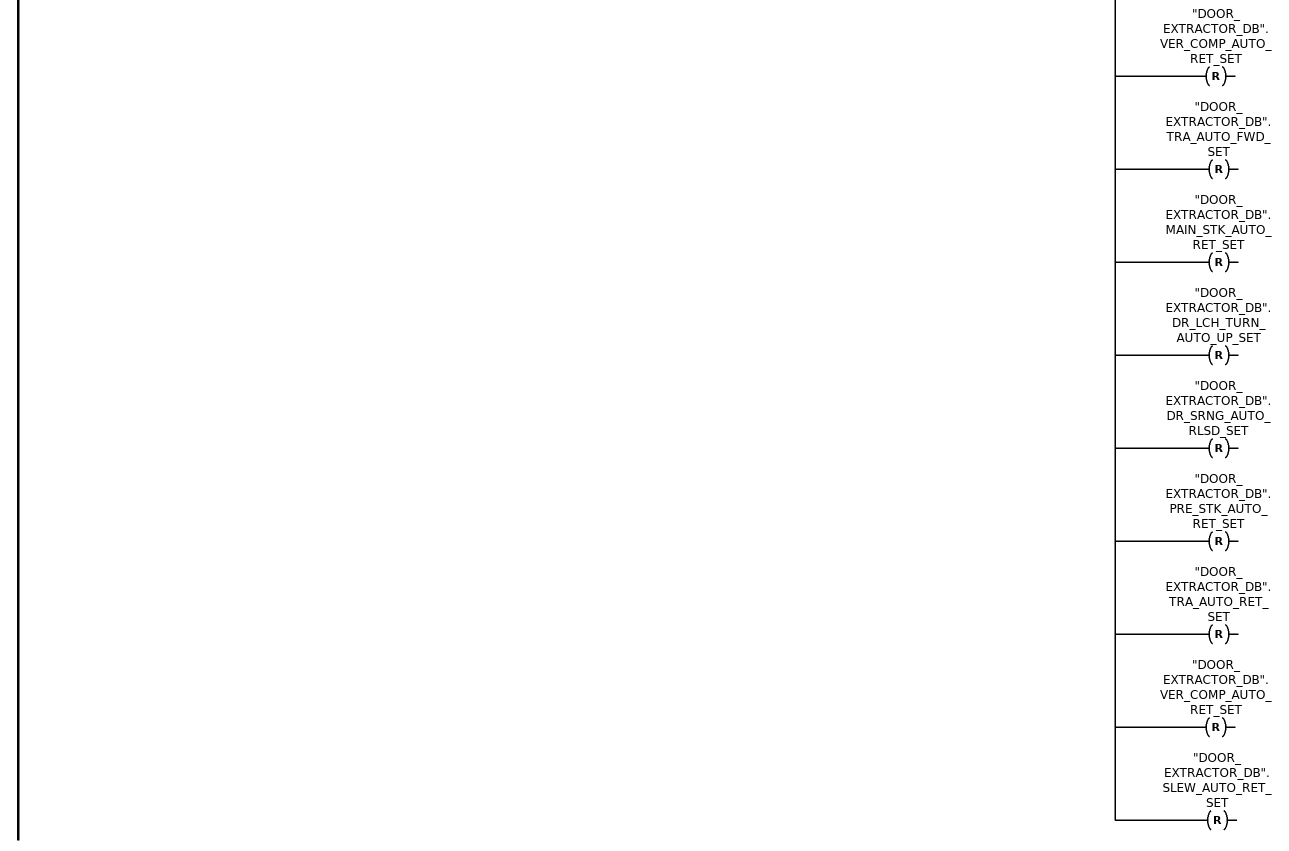
NETWORK
TITLE =
      A     "ALWAYS_ON";
      A     "DOOR_EXTRACTOR_DB".SLEW_NR_FWD_OP_CUT;
      A(;
      O     "DOOR_EXTRACTOR_DB".VER_COMP_RET_OP_CUT;
      O     "ALWAYS_ON";
      );
      A     "DOOR_EXTRACTOR_DB".TRA_NOR_RET_OP_CUT;
      A     "DOOR_EXTRACTOR_DB".PRE_STK_UP_OP_CUT;
      A     "DOOR_EXTRACTOR_DB".DR_SPNG_LK_OP_CUT;
      A     "DOOR_EXTRACTOR_DB".DR_LCH_DN_OP_CUT;
      A     "DOOR_EXTRACTOR_DB".MAIN_STK_UP_OP_CUT;
      A     "DOOR_EXTRACTOR_DB".FIN_STK_UP_OP_CUT;
      =     "DOOR_EXTRACTOR_DB".DR_EXT_AUTO_OPER_FIN;
      R     "DOOR_EXTRACTOR_DB".SLEW_AUTO_FWD_SET;
      R     "DOOR_EXTRACTOR_DB".VER_COMP_AUTO_FWD_SET;
      R     "DOOR_EXTRACTOR_DB".TRA_AUTO_FWD_SET;
      R     "DOOR_EXTRACTOR_DB".PRE_STK_AUTO_FWD_SET;
      R     "DOOR_EXTRACTOR_DB".DR_SPNG_AUTO_PRSD_SET;
      R     "DOOR_EXTRACTOR_DB".DR_LCH_TURN_AUTO_DN_SET;
      R     "DOOR_EXTRACTOR_DB".MAIN_STK_AUTO_FWD_SET;
      R     "DOOR_EXTRACTOR_DB".TRA_AUTO_RET_SET;
      R     "DOOR_EXTRACTOR_DB".VER_COMP_AUTO_RET_SET;
      R     "DOOR_EXTRACTOR_DB".FIN_STK_AUTO_FWD_SET;
      R     "DOOR_EXTRACTOR_DB".SLEW_AUTO_RET_SET;
      R     "DOOR_EXTRACTOR_DB".SLEW_AUTO_FWD_SET;
      R     "DOOR_EXTRACTOR_DB".FIN_STK_AUTO_RET_SET;
      R     "DOOR_EXTRACTOR_DB".VER_COMP_AUTO_RET_SET;
      R     "DOOR_EXTRACTOR_DB".TRA_AUTO_FWD_SET;
      R     "DOOR_EXTRACTOR_DB".MAIN_STK_AUTO_RET_SET;
      R     "DOOR_EXTRACTOR_DB".DR_LCH_TURN_AUTO_UP_SET;
      R     "DOOR_EXTRACTOR_DB".DR_SRNG_AUTO_RLSD_SET;
      R     "DOOR_EXTRACTOR_DB".PRE_STK_AUTO_RET_SET;
      R     "DOOR_EXTRACTOR_DB".TRA_AUTO_RET_SET;
      R     "DOOR_EXTRACTOR_DB".VER_COMP_AUTO_RET_SET;
      R     "DOOR_EXTRACTOR_DB".SLEW_AUTO_RET_SET;
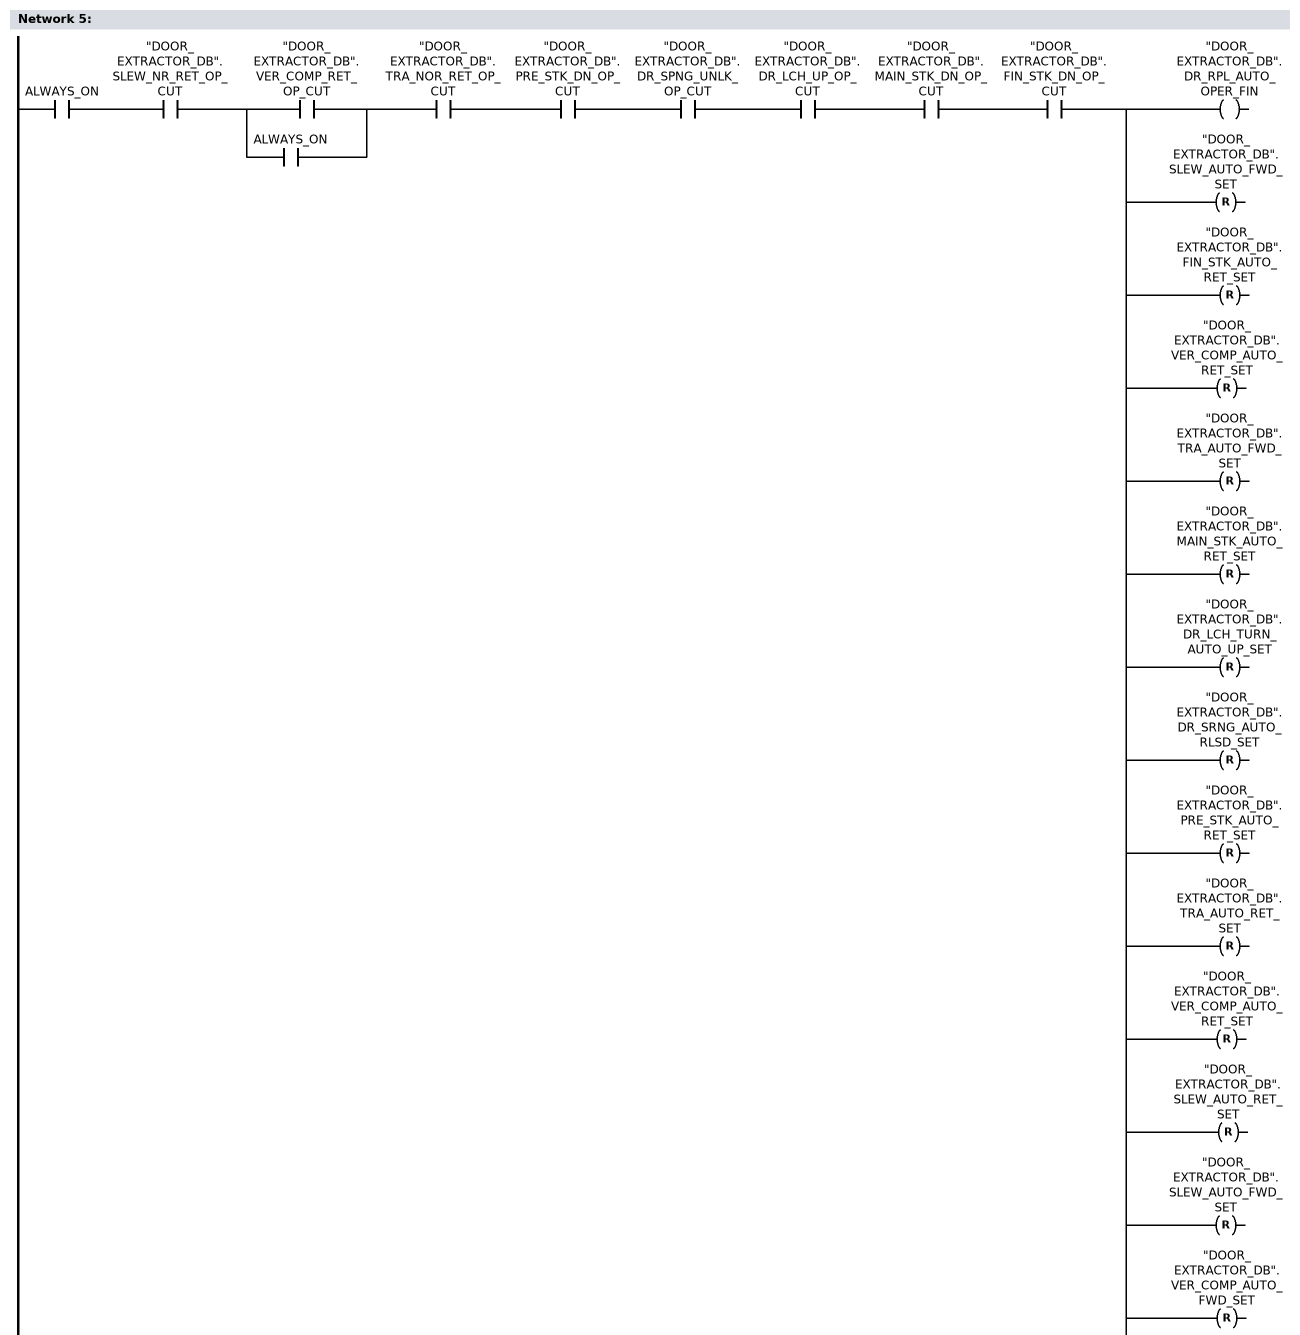
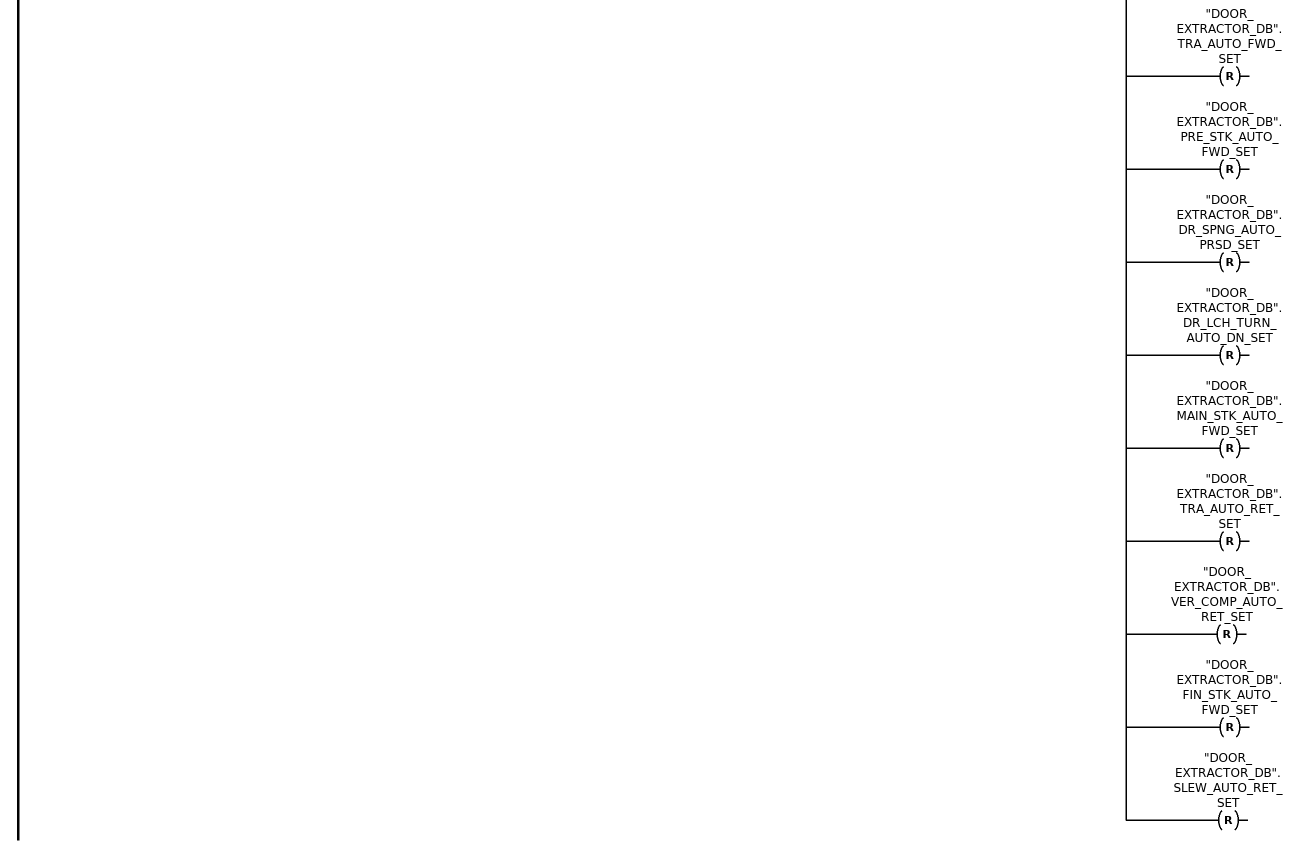
NETWORK
TITLE =
      A     "ALWAYS_ON";
      A     "DOOR_EXTRACTOR_DB".SLEW_NR_RET_OP_CUT;
      A(;
      O     "DOOR_EXTRACTOR_DB".VER_COMP_RET_OP_CUT;
      O     "ALWAYS_ON";
      );
      A     "DOOR_EXTRACTOR_DB".TRA_NOR_RET_OP_CUT;
      A     "DOOR_EXTRACTOR_DB".PRE_STK_DN_OP_CUT;
      A     "DOOR_EXTRACTOR_DB".DR_SPNG_UNLK_OP_CUT;
      A     "DOOR_EXTRACTOR_DB".DR_LCH_UP_OP_CUT;
      A     "DOOR_EXTRACTOR_DB".MAIN_STK_DN_OP_CUT;
      A     "DOOR_EXTRACTOR_DB".FIN_STK_DN_OP_CUT;
      =     "DOOR_EXTRACTOR_DB".DR_RPL_AUTO_OPER_FIN;
      R     "DOOR_EXTRACTOR_DB".SLEW_AUTO_FWD_SET;
      R     "DOOR_EXTRACTOR_DB".FIN_STK_AUTO_RET_SET;
      R     "DOOR_EXTRACTOR_DB".VER_COMP_AUTO_RET_SET;
      R     "DOOR_EXTRACTOR_DB".TRA_AUTO_FWD_SET;
      R     "DOOR_EXTRACTOR_DB".MAIN_STK_AUTO_RET_SET;
      R     "DOOR_EXTRACTOR_DB".DR_LCH_TURN_AUTO_UP_SET;
      R     "DOOR_EXTRACTOR_DB".DR_SRNG_AUTO_RLSD_SET;
      R     "DOOR_EXTRACTOR_DB".PRE_STK_AUTO_RET_SET;
      R     "DOOR_EXTRACTOR_DB".TRA_AUTO_RET_SET;
      R     "DOOR_EXTRACTOR_DB".VER_COMP_AUTO_RET_SET;
      R     "DOOR_EXTRACTOR_DB".SLEW_AUTO_RET_SET;
      R     "DOOR_EXTRACTOR_DB".SLEW_AUTO_FWD_SET;
      R     "DOOR_EXTRACTOR_DB".VER_COMP_AUTO_FWD_SET;
      R     "DOOR_EXTRACTOR_DB".TRA_AUTO_FWD_SET;
      R     "DOOR_EXTRACTOR_DB".PRE_STK_AUTO_FWD_SET;
      R     "DOOR_EXTRACTOR_DB".DR_SPNG_AUTO_PRSD_SET;
      R     "DOOR_EXTRACTOR_DB".DR_LCH_TURN_AUTO_DN_SET;
      R     "DOOR_EXTRACTOR_DB".MAIN_STK_AUTO_FWD_SET;
      R     "DOOR_EXTRACTOR_DB".TRA_AUTO_RET_SET;
      R     "DOOR_EXTRACTOR_DB".VER_COMP_AUTO_RET_SET;
      R     "DOOR_EXTRACTOR_DB".FIN_STK_AUTO_FWD_SET;
      R     "DOOR_EXTRACTOR_DB".SLEW_AUTO_RET_SET;
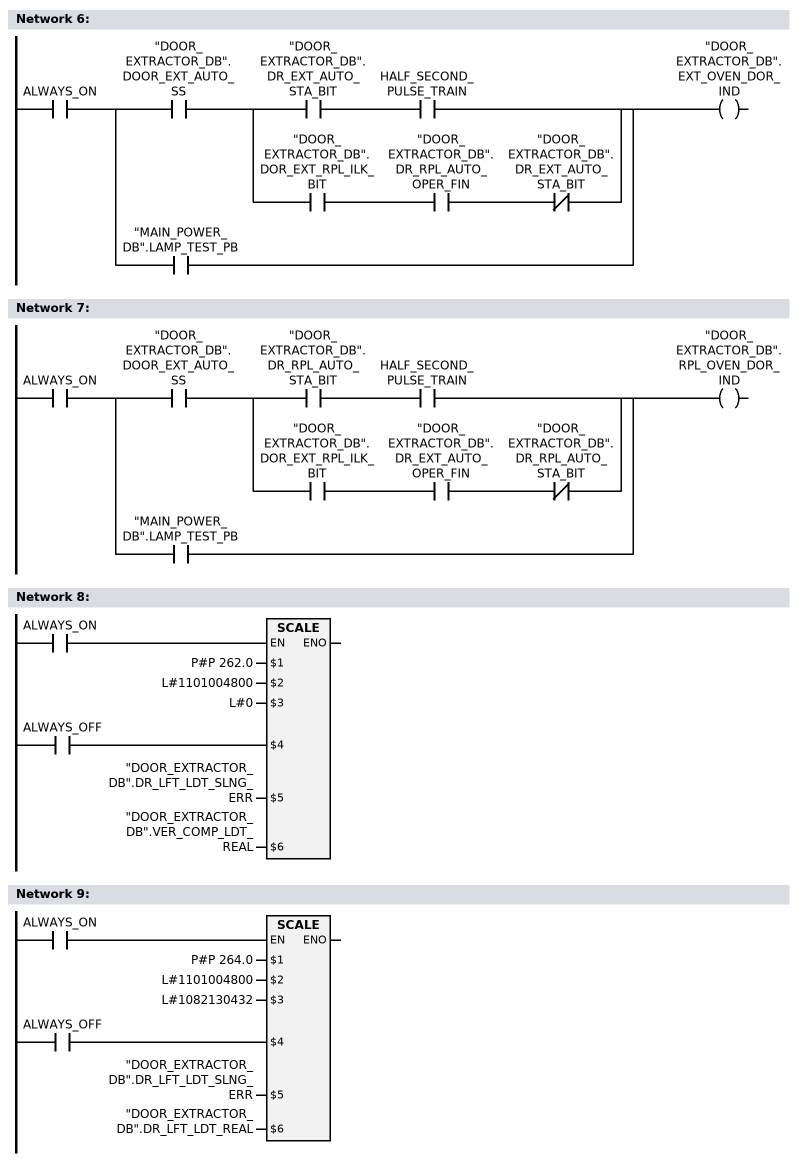
NETWORK
TITLE =
      A     "ALWAYS_ON";
      A(;
      A     "DOOR_EXTRACTOR_DB".DOOR_EXT_AUTO_SS;
      A(;
      A     "DOOR_EXTRACTOR_DB".DR_EXT_AUTO_STA_BIT;
      A     "HALF_SECOND_PULSE_TRAIN";
      O;
      A     "DOOR_EXTRACTOR_DB".DOR_EXT_RPL_ILK_BIT;
      A     "DOOR_EXTRACTOR_DB".DR_RPL_AUTO_OPER_FIN;
      AN    "DOOR_EXTRACTOR_DB".DR_EXT_AUTO_STA_BIT;
      );
      O     "MAIN_POWER_DB".LAMP_TEST_PB;
      );
      =     "DOOR_EXTRACTOR_DB".EXT_OVEN_DOR_IND;
NETWORK
TITLE =
      A     "ALWAYS_ON";
      A(;
      A     "DOOR_EXTRACTOR_DB".DOOR_EXT_AUTO_SS;
      A(;
      A     "DOOR_EXTRACTOR_DB".DR_RPL_AUTO_STA_BIT;
      A     "HALF_SECOND_PULSE_TRAIN";
      O;
      A     "DOOR_EXTRACTOR_DB".DOR_EXT_RPL_ILK_BIT;
      A     "DOOR_EXTRACTOR_DB".DR_EXT_AUTO_OPER_FIN;
      AN    "DOOR_EXTRACTOR_DB".DR_RPL_AUTO_STA_BIT;
      );
      O     "MAIN_POWER_DB".LAMP_TEST_PB;
      );
      =     "DOOR_EXTRACTOR_DB".RPL_OVEN_DOR_IND;
NETWORK
TITLE =
      A     "ALWAYS_OFF";
      =     L 0.0;
      BLD   103;
      A     "ALWAYS_ON";
      JNB   M001;
      CALL  "SCALE" (
           $1                       := P#P 262.0,
           $2                       := L#1101004800,
           $3                       := L#0,
           $4                       := L 0.0,
           $5                       := "DOOR_EXTRACTOR_DB".DR_LFT_LDT_SLNG_ERR,
           $6                       := "DOOR_EXTRACTOR_DB".VER_COMP_LDT_REAL);
M001: NOP   0;
NETWORK
TITLE =
      A     "ALWAYS_OFF";
      =     L 0.0;
      BLD   103;
      A     "ALWAYS_ON";
      JNB   M002;
      CALL  "SCALE" (
           $1                       := P#P 264.0,
           $2                       := L#1101004800,
           $3                       := L#1082130432,
           $4                       := L 0.0,
           $5                       := "DOOR_EXTRACTOR_DB".DR_LFT_LDT_SLNG_ERR,
           $6                       := "DOOR_EXTRACTOR_DB".DR_LFT_LDT_REAL);
M002: NOP   0;
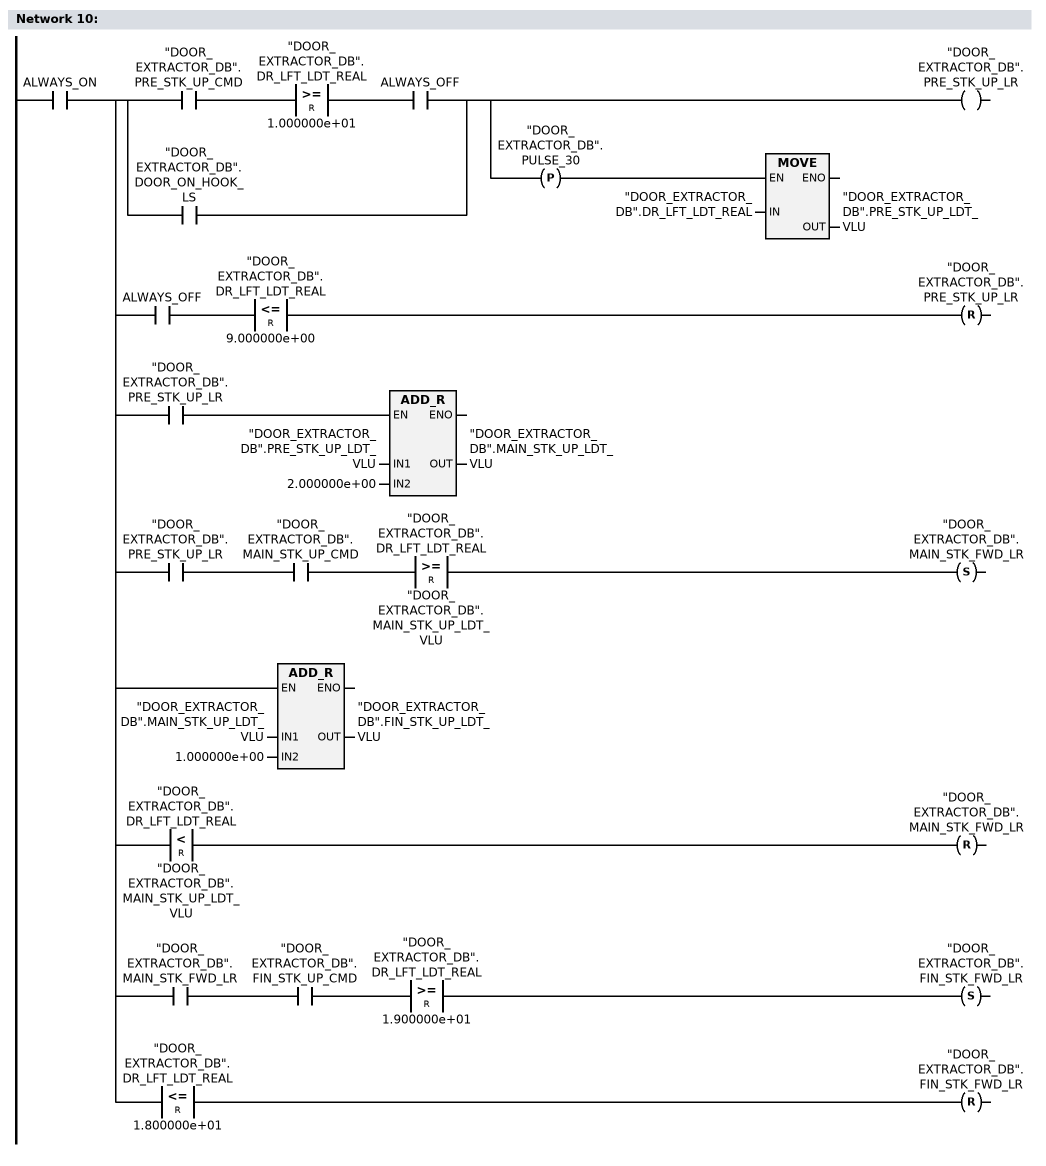
NETWORK
TITLE =
      A     "ALWAYS_ON";
      =     L 0.0;
      A     L 0.0;
      A(;
      A     "DOOR_EXTRACTOR_DB".PRE_STK_UP_CMD;
      A(;
      L     "DOOR_EXTRACTOR_DB".DR_LFT_LDT_REAL;
      L     1.000000e+01;
      >=R;
      );
      A     "ALWAYS_OFF";
      O     "DOOR_EXTRACTOR_DB".DOOR_ON_HOOK_LS;
      );
      =     L 0.1;
      A     L 0.1;
      BLD   102;
      =     "DOOR_EXTRACTOR_DB".PRE_STK_UP_LR;
      A     L 0.1;
      FP    "DOOR_EXTRACTOR_DB".PULSE_30;
      JNB   M003;
      L     "DOOR_EXTRACTOR_DB".DR_LFT_LDT_REAL;
      T     "DOOR_EXTRACTOR_DB".PRE_STK_UP_LDT_VLU;
M003: NOP   0;
      A     L 0.0;
      A     "ALWAYS_OFF";
      A(;
      L     "DOOR_EXTRACTOR_DB".DR_LFT_LDT_REAL;
      L     9.000000e+00;
      <=R;
      );
      R     "DOOR_EXTRACTOR_DB".PRE_STK_UP_LR;
      A     L 0.0;
      A     "DOOR_EXTRACTOR_DB".PRE_STK_UP_LR;
      JNB   M004;
      L     "DOOR_EXTRACTOR_DB".PRE_STK_UP_LDT_VLU;
      L     2.000000e+00;
      +R;
      T     "DOOR_EXTRACTOR_DB".MAIN_STK_UP_LDT_VLU;
M004: NOP   0;
      A     L 0.0;
      A     "DOOR_EXTRACTOR_DB".PRE_STK_UP_LR;
      A     "DOOR_EXTRACTOR_DB".MAIN_STK_UP_CMD;
      A(;
      L     "DOOR_EXTRACTOR_DB".DR_LFT_LDT_REAL;
      L     "DOOR_EXTRACTOR_DB".MAIN_STK_UP_LDT_VLU;
      >=R;
      );
      S     "DOOR_EXTRACTOR_DB".MAIN_STK_FWD_LR;
      A     L 0.0;
      JNB   M005;
      L     "DOOR_EXTRACTOR_DB".MAIN_STK_UP_LDT_VLU;
      L     1.000000e+00;
      +R;
      T     "DOOR_EXTRACTOR_DB".FIN_STK_UP_LDT_VLU;
M005: NOP   0;
      A     L 0.0;
      A(;
      L     "DOOR_EXTRACTOR_DB".DR_LFT_LDT_REAL;
      L     "DOOR_EXTRACTOR_DB".MAIN_STK_UP_LDT_VLU;
      <R;
      );
      R     "DOOR_EXTRACTOR_DB".MAIN_STK_FWD_LR;
      A     L 0.0;
      A     "DOOR_EXTRACTOR_DB".MAIN_STK_FWD_LR;
      A     "DOOR_EXTRACTOR_DB".FIN_STK_UP_CMD;
      A(;
      L     "DOOR_EXTRACTOR_DB".DR_LFT_LDT_REAL;
      L     1.900000e+01;
      >=R;
      );
      S     "DOOR_EXTRACTOR_DB".FIN_STK_FWD_LR;
      A     L 0.0;
      A(;
      L     "DOOR_EXTRACTOR_DB".DR_LFT_LDT_REAL;
      L     1.800000e+01;
      <=R;
      );
      R     "DOOR_EXTRACTOR_DB".FIN_STK_FWD_LR;
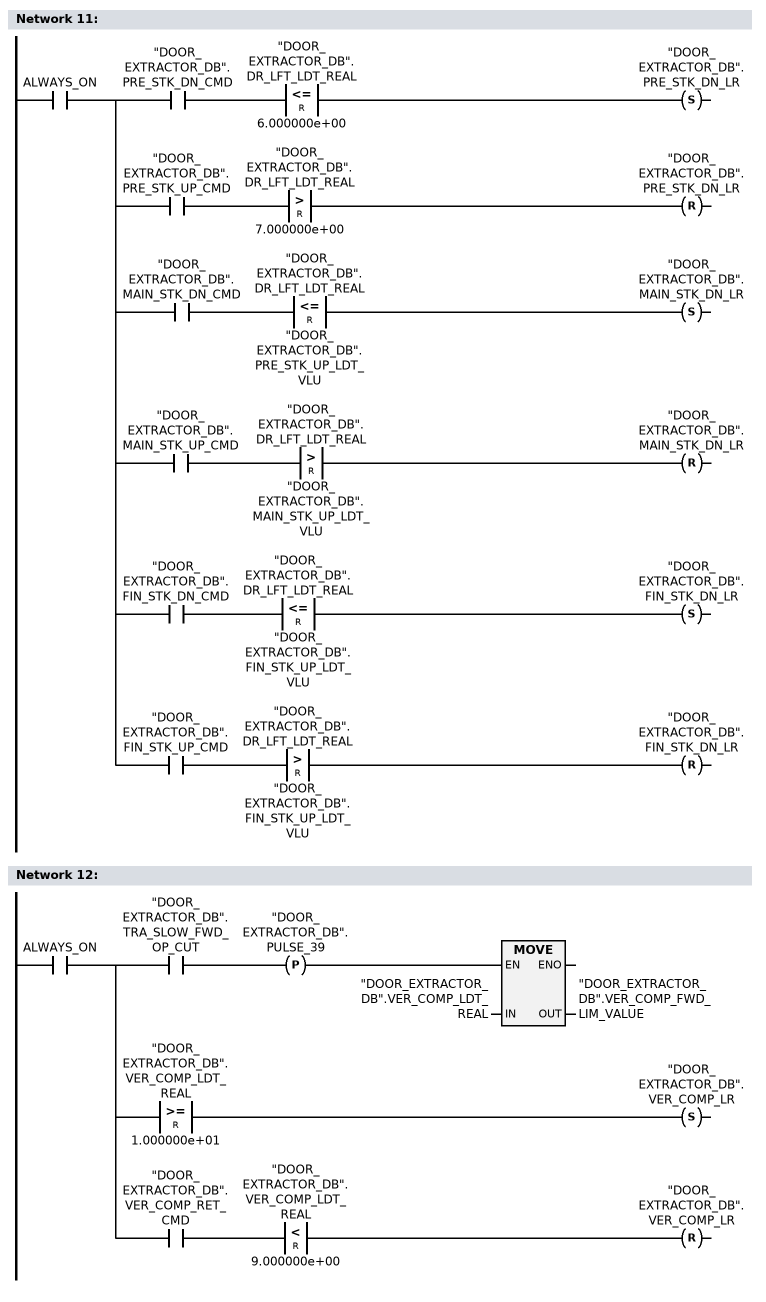
NETWORK
TITLE =
      A     "ALWAYS_ON";
      =     L 0.0;
      A     L 0.0;
      A     "DOOR_EXTRACTOR_DB".PRE_STK_DN_CMD;
      A(;
      L     "DOOR_EXTRACTOR_DB".DR_LFT_LDT_REAL;
      L     6.000000e+00;
      <=R;
      );
      S     "DOOR_EXTRACTOR_DB".PRE_STK_DN_LR;
      A     L 0.0;
      A     "DOOR_EXTRACTOR_DB".PRE_STK_UP_CMD;
      A(;
      L     "DOOR_EXTRACTOR_DB".DR_LFT_LDT_REAL;
      L     7.000000e+00;
      >R;
      );
      R     "DOOR_EXTRACTOR_DB".PRE_STK_DN_LR;
      A     L 0.0;
      A     "DOOR_EXTRACTOR_DB".MAIN_STK_DN_CMD;
      A(;
      L     "DOOR_EXTRACTOR_DB".DR_LFT_LDT_REAL;
      L     "DOOR_EXTRACTOR_DB".PRE_STK_UP_LDT_VLU;
      <=R;
      );
      S     "DOOR_EXTRACTOR_DB".MAIN_STK_DN_LR;
      A     L 0.0;
      A     "DOOR_EXTRACTOR_DB".MAIN_STK_UP_CMD;
      A(;
      L     "DOOR_EXTRACTOR_DB".DR_LFT_LDT_REAL;
      L     "DOOR_EXTRACTOR_DB".MAIN_STK_UP_LDT_VLU;
      >R;
      );
      R     "DOOR_EXTRACTOR_DB".MAIN_STK_DN_LR;
      A     L 0.0;
      A     "DOOR_EXTRACTOR_DB".FIN_STK_DN_CMD;
      A(;
      L     "DOOR_EXTRACTOR_DB".DR_LFT_LDT_REAL;
      L     "DOOR_EXTRACTOR_DB".FIN_STK_UP_LDT_VLU;
      <=R;
      );
      S     "DOOR_EXTRACTOR_DB".FIN_STK_DN_LR;
      A     L 0.0;
      A     "DOOR_EXTRACTOR_DB".FIN_STK_UP_CMD;
      A(;
      L     "DOOR_EXTRACTOR_DB".DR_LFT_LDT_REAL;
      L     "DOOR_EXTRACTOR_DB".FIN_STK_UP_LDT_VLU;
      >R;
      );
      R     "DOOR_EXTRACTOR_DB".FIN_STK_DN_LR;
NETWORK
TITLE =
      A     "ALWAYS_ON";
      =     L 0.0;
      A     L 0.0;
      A     "DOOR_EXTRACTOR_DB".TRA_SLOW_FWD_OP_CUT;
      FP    "DOOR_EXTRACTOR_DB".PULSE_39;
      JNB   M006;
      L     "DOOR_EXTRACTOR_DB".VER_COMP_LDT_REAL;
      T     "DOOR_EXTRACTOR_DB".VER_COMP_FWD_LIM_VALUE;
M006: NOP   0;
      A     L 0.0;
      A(;
      L     "DOOR_EXTRACTOR_DB".VER_COMP_LDT_REAL;
      L     1.000000e+01;
      >=R;
      );
      S     "DOOR_EXTRACTOR_DB".VER_COMP_LR;
      A     L 0.0;
      A     "DOOR_EXTRACTOR_DB".VER_COMP_RET_CMD;
      A(;
      L     "DOOR_EXTRACTOR_DB".VER_COMP_LDT_REAL;
      L     9.000000e+00;
      <R;
      );
      R     "DOOR_EXTRACTOR_DB".VER_COMP_LR;
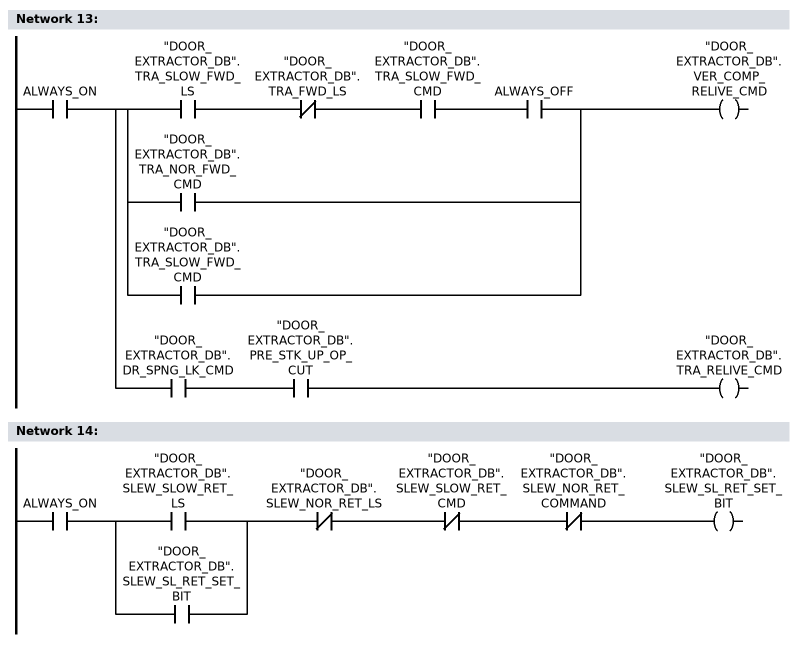
NETWORK
TITLE =
      A     "ALWAYS_ON";
      =     L 0.0;
      A     L 0.0;
      A(;
      A     "DOOR_EXTRACTOR_DB".TRA_SLOW_FWD_LS;
      AN    "DOOR_EXTRACTOR_DB".TRA_FWD_LS;
      A     "DOOR_EXTRACTOR_DB".TRA_SLOW_FWD_CMD;
      A     "ALWAYS_OFF";
      O     "DOOR_EXTRACTOR_DB".TRA_NOR_FWD_CMD;
      O     "DOOR_EXTRACTOR_DB".TRA_SLOW_FWD_CMD;
      );
      =     "DOOR_EXTRACTOR_DB".VER_COMP_RELIVE_CMD;
      A     L 0.0;
      A     "DOOR_EXTRACTOR_DB".DR_SPNG_LK_CMD;
      A     "DOOR_EXTRACTOR_DB".PRE_STK_UP_OP_CUT;
      =     "DOOR_EXTRACTOR_DB".TRA_RELIVE_CMD;
NETWORK
TITLE =
      A     "ALWAYS_ON";
      A(;
      O     "DOOR_EXTRACTOR_DB".SLEW_SLOW_RET_LS;
      O     "DOOR_EXTRACTOR_DB".SLEW_SL_RET_SET_BIT;
      );
      AN    "DOOR_EXTRACTOR_DB".SLEW_NOR_RET_LS;
      AN    "DOOR_EXTRACTOR_DB".SLEW_SLOW_RET_CMD;
      AN    "DOOR_EXTRACTOR_DB".SLEW_NOR_RET_COMMAND;
      =     "DOOR_EXTRACTOR_DB".SLEW_SL_RET_SET_BIT;
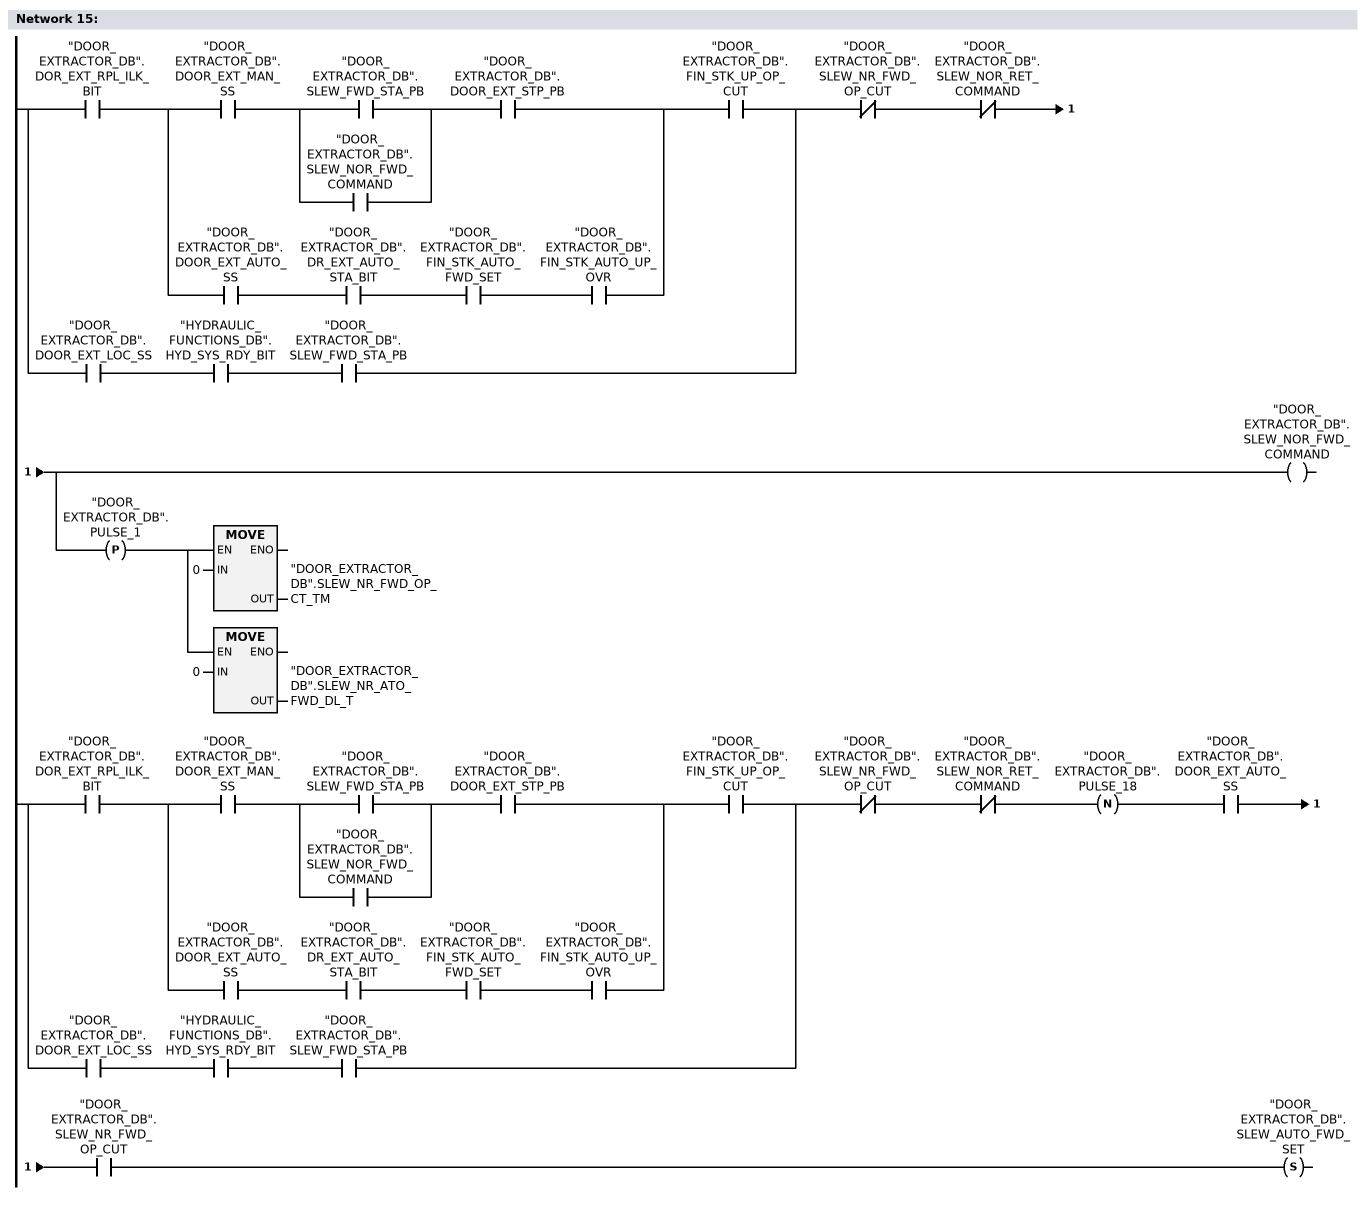
NETWORK
TITLE =
      A(;
      A     "DOOR_EXTRACTOR_DB".DOR_EXT_RPL_ILK_BIT;
      A(;
      A     "DOOR_EXTRACTOR_DB".DOOR_EXT_MAN_SS;
      A(;
      O     "DOOR_EXTRACTOR_DB".SLEW_FWD_STA_PB;
      O     "DOOR_EXTRACTOR_DB".SLEW_NOR_FWD_COMMAND;
      );
      A     "DOOR_EXTRACTOR_DB".DOOR_EXT_STP_PB;
      O;
      A     "DOOR_EXTRACTOR_DB".DOOR_EXT_AUTO_SS;
      A     "DOOR_EXTRACTOR_DB".DR_EXT_AUTO_STA_BIT;
      A     "DOOR_EXTRACTOR_DB".FIN_STK_AUTO_FWD_SET;
      A     "DOOR_EXTRACTOR_DB".FIN_STK_AUTO_UP_OVR;
      );
      A     "DOOR_EXTRACTOR_DB".FIN_STK_UP_OP_CUT;
      O;
      A     "DOOR_EXTRACTOR_DB".DOOR_EXT_LOC_SS;
      A     "HYDRAULIC_FUNCTIONS_DB".HYD_SYS_RDY_BIT;
      A     "DOOR_EXTRACTOR_DB".SLEW_FWD_STA_PB;
      );
      AN    "DOOR_EXTRACTOR_DB".SLEW_NR_FWD_OP_CUT;
      AN    "DOOR_EXTRACTOR_DB".SLEW_NOR_RET_COMMAND;
      =     L 0.0;
      A     L 0.0;
      BLD   102;
      =     "DOOR_EXTRACTOR_DB".SLEW_NOR_FWD_COMMAND;
      A(;
      A     L 0.0;
      FN    "DOOR_EXTRACTOR_DB".PULSE_18;
      );
      A     "DOOR_EXTRACTOR_DB".DOOR_EXT_AUTO_SS;
      A     "DOOR_EXTRACTOR_DB".SLEW_NR_FWD_OP_CUT;
      S     "DOOR_EXTRACTOR_DB".SLEW_AUTO_FWD_SET;
      A     L 0.0;
      FP    "DOOR_EXTRACTOR_DB".PULSE_1;
      =     L 0.1;
      A     L 0.1;
      JNB   M007;
      L     0;
      T     "DOOR_EXTRACTOR_DB".SLEW_NR_FWD_OP_CT_TM;
M007: NOP   0;
      A     L 0.1;
      JNB   M008;
      L     0;
      T     "DOOR_EXTRACTOR_DB".SLEW_NR_ATO_FWD_DL_T;
M008: NOP   0;
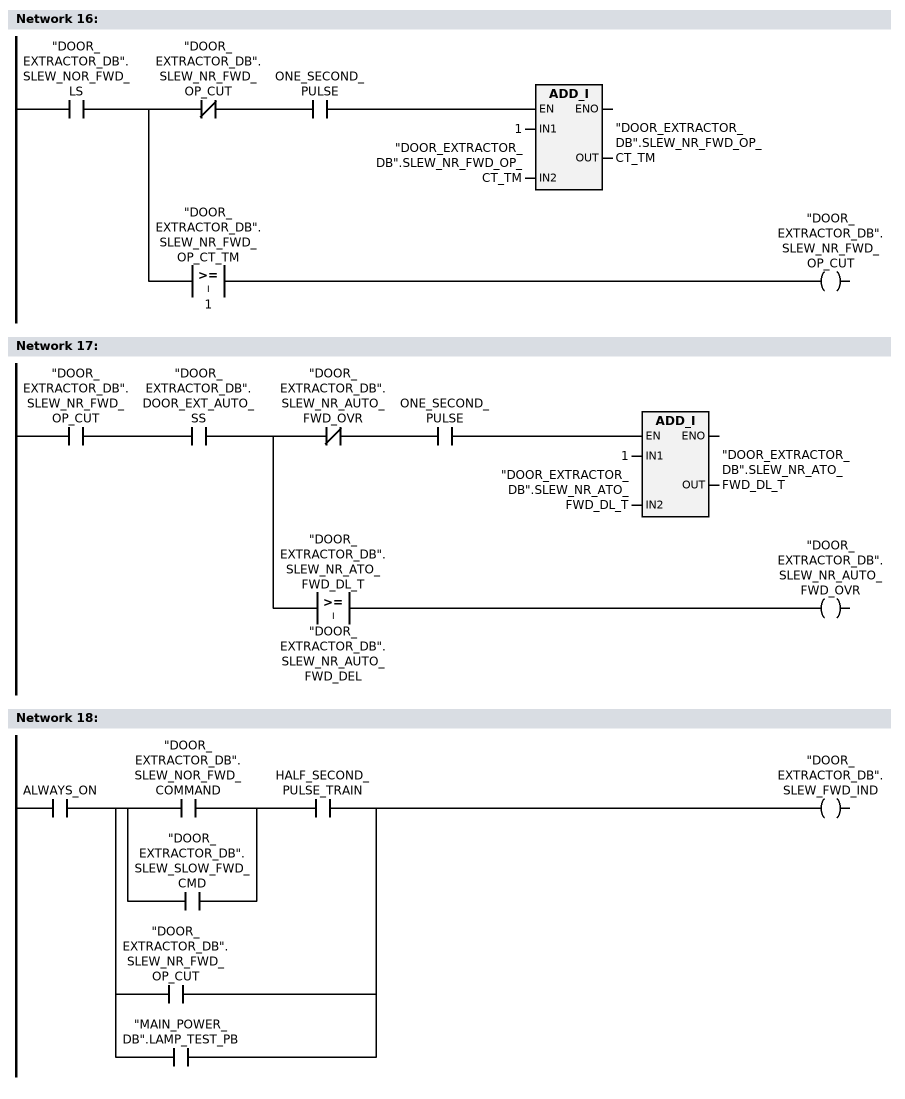
NETWORK
TITLE =
      A     "DOOR_EXTRACTOR_DB".SLEW_NOR_FWD_LS;
      =     L 0.0;
      A     L 0.0;
      AN    "DOOR_EXTRACTOR_DB".SLEW_NR_FWD_OP_CUT;
      A     "ONE_SECOND_PULSE";
      JNB   M009;
      L     1;
      L     "DOOR_EXTRACTOR_DB".SLEW_NR_FWD_OP_CT_TM;
      +I;
      T     "DOOR_EXTRACTOR_DB".SLEW_NR_FWD_OP_CT_TM;
M009: NOP   0;
      A     L 0.0;
      A(;
      L     "DOOR_EXTRACTOR_DB".SLEW_NR_FWD_OP_CT_TM;
      L     1;
      >=I;
      );
      =     "DOOR_EXTRACTOR_DB".SLEW_NR_FWD_OP_CUT;
NETWORK
TITLE =
      A     "DOOR_EXTRACTOR_DB".SLEW_NR_FWD_OP_CUT;
      A     "DOOR_EXTRACTOR_DB".DOOR_EXT_AUTO_SS;
      =     L 0.0;
      A     L 0.0;
      AN    "DOOR_EXTRACTOR_DB".SLEW_NR_AUTO_FWD_OVR;
      A     "ONE_SECOND_PULSE";
      JNB   M010;
      L     1;
      L     "DOOR_EXTRACTOR_DB".SLEW_NR_ATO_FWD_DL_T;
      +I;
      T     "DOOR_EXTRACTOR_DB".SLEW_NR_ATO_FWD_DL_T;
M010: NOP   0;
      A     L 0.0;
      A(;
      L     "DOOR_EXTRACTOR_DB".SLEW_NR_ATO_FWD_DL_T;
      L     "DOOR_EXTRACTOR_DB".SLEW_NR_AUTO_FWD_DEL;
      >=I;
      );
      =     "DOOR_EXTRACTOR_DB".SLEW_NR_AUTO_FWD_OVR;
NETWORK
TITLE =
      A     "ALWAYS_ON";
      A(;
      A(;
      O     "DOOR_EXTRACTOR_DB".SLEW_NOR_FWD_COMMAND;
      O     "DOOR_EXTRACTOR_DB".SLEW_SLOW_FWD_CMD;
      );
      A     "HALF_SECOND_PULSE_TRAIN";
      O     "DOOR_EXTRACTOR_DB".SLEW_NR_FWD_OP_CUT;
      O     "MAIN_POWER_DB".LAMP_TEST_PB;
      );
      =     "DOOR_EXTRACTOR_DB".SLEW_FWD_IND;
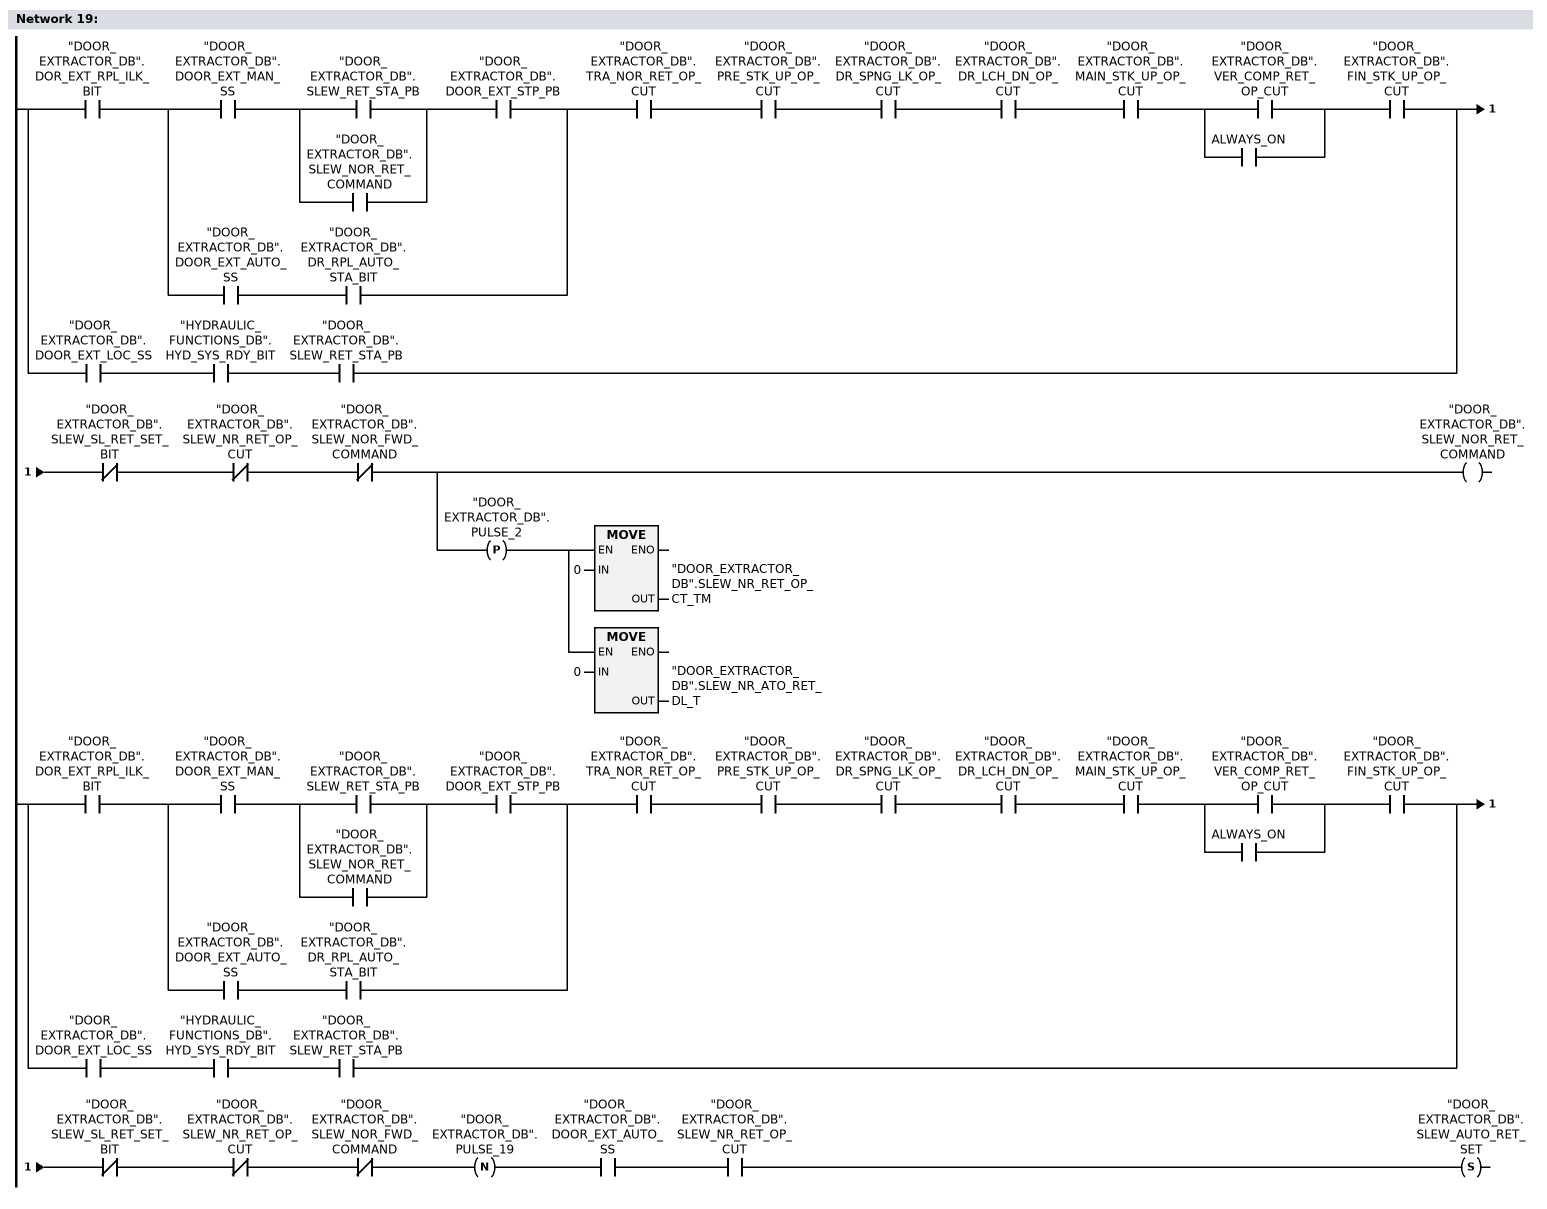
NETWORK
TITLE =
      A(;
      A     "DOOR_EXTRACTOR_DB".DOR_EXT_RPL_ILK_BIT;
      A(;
      A     "DOOR_EXTRACTOR_DB".DOOR_EXT_MAN_SS;
      A(;
      O     "DOOR_EXTRACTOR_DB".SLEW_RET_STA_PB;
      O     "DOOR_EXTRACTOR_DB".SLEW_NOR_RET_COMMAND;
      );
      A     "DOOR_EXTRACTOR_DB".DOOR_EXT_STP_PB;
      O;
      A     "DOOR_EXTRACTOR_DB".DOOR_EXT_AUTO_SS;
      A     "DOOR_EXTRACTOR_DB".DR_RPL_AUTO_STA_BIT;
      );
      A     "DOOR_EXTRACTOR_DB".TRA_NOR_RET_OP_CUT;
      A     "DOOR_EXTRACTOR_DB".PRE_STK_UP_OP_CUT;
      A     "DOOR_EXTRACTOR_DB".DR_SPNG_LK_OP_CUT;
      A     "DOOR_EXTRACTOR_DB".DR_LCH_DN_OP_CUT;
      A     "DOOR_EXTRACTOR_DB".MAIN_STK_UP_OP_CUT;
      A(;
      O     "DOOR_EXTRACTOR_DB".VER_COMP_RET_OP_CUT;
      O     "ALWAYS_ON";
      );
      A     "DOOR_EXTRACTOR_DB".FIN_STK_UP_OP_CUT;
      O;
      A     "DOOR_EXTRACTOR_DB".DOOR_EXT_LOC_SS;
      A     "HYDRAULIC_FUNCTIONS_DB".HYD_SYS_RDY_BIT;
      A     "DOOR_EXTRACTOR_DB".SLEW_RET_STA_PB;
      );
      AN    "DOOR_EXTRACTOR_DB".SLEW_SL_RET_SET_BIT;
      AN    "DOOR_EXTRACTOR_DB".SLEW_NR_RET_OP_CUT;
      AN    "DOOR_EXTRACTOR_DB".SLEW_NOR_FWD_COMMAND;
      =     L 0.0;
      A     L 0.0;
      BLD   102;
      =     "DOOR_EXTRACTOR_DB".SLEW_NOR_RET_COMMAND;
      A(;
      A     L 0.0;
      FN    "DOOR_EXTRACTOR_DB".PULSE_19;
      );
      A     "DOOR_EXTRACTOR_DB".DOOR_EXT_AUTO_SS;
      A     "DOOR_EXTRACTOR_DB".SLEW_NR_RET_OP_CUT;
      S     "DOOR_EXTRACTOR_DB".SLEW_AUTO_RET_SET;
      A     L 0.0;
      FP    "DOOR_EXTRACTOR_DB".PULSE_2;
      =     L 0.1;
      A     L 0.1;
      JNB   M011;
      L     0;
      T     "DOOR_EXTRACTOR_DB".SLEW_NR_RET_OP_CT_TM;
M011: NOP   0;
      A     L 0.1;
      JNB   M012;
      L     0;
      T     "DOOR_EXTRACTOR_DB".SLEW_NR_ATO_RET_DL_T;
M012: NOP   0;
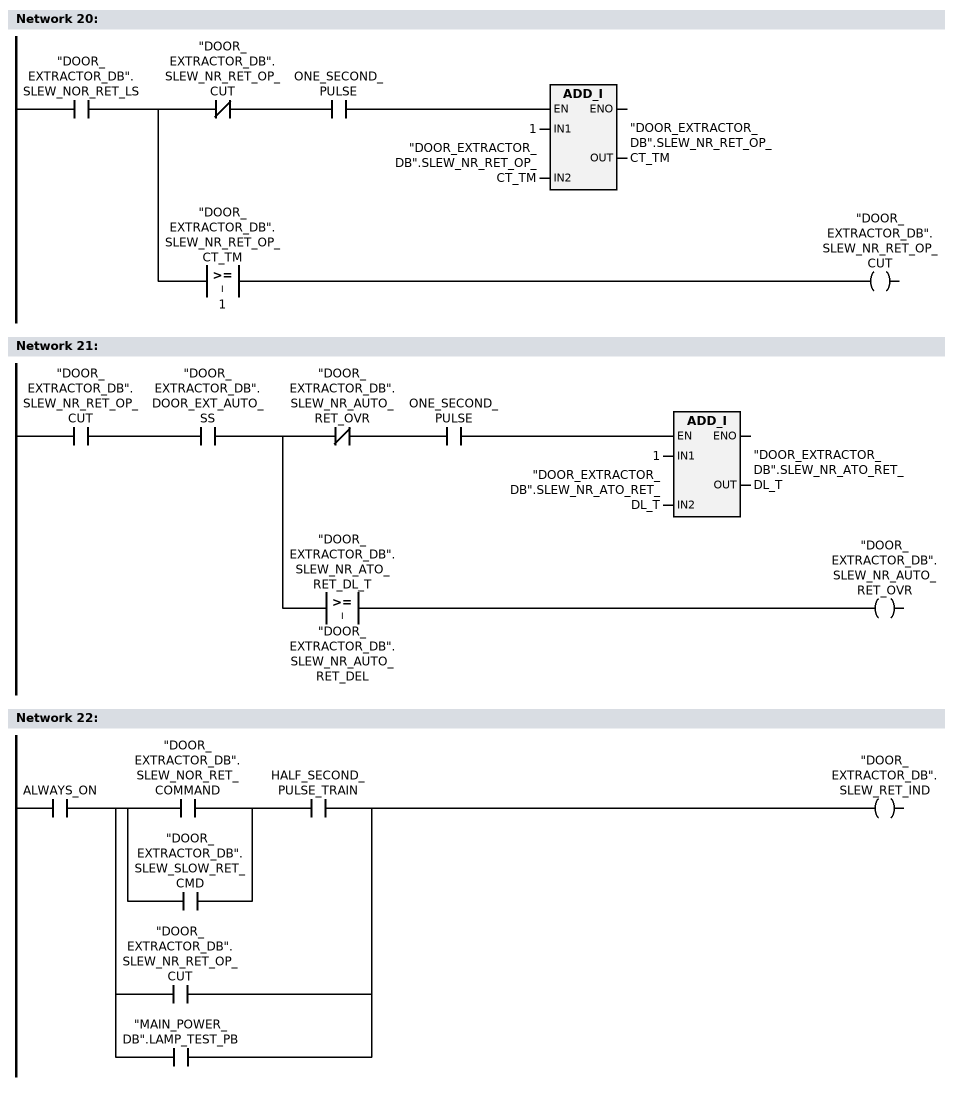
NETWORK
TITLE =
      A     "DOOR_EXTRACTOR_DB".SLEW_NOR_RET_LS;
      =     L 0.0;
      A     L 0.0;
      AN    "DOOR_EXTRACTOR_DB".SLEW_NR_RET_OP_CUT;
      A     "ONE_SECOND_PULSE";
      JNB   M013;
      L     1;
      L     "DOOR_EXTRACTOR_DB".SLEW_NR_RET_OP_CT_TM;
      +I;
      T     "DOOR_EXTRACTOR_DB".SLEW_NR_RET_OP_CT_TM;
M013: NOP   0;
      A     L 0.0;
      A(;
      L     "DOOR_EXTRACTOR_DB".SLEW_NR_RET_OP_CT_TM;
      L     1;
      >=I;
      );
      =     "DOOR_EXTRACTOR_DB".SLEW_NR_RET_OP_CUT;
NETWORK
TITLE =
      A     "DOOR_EXTRACTOR_DB".SLEW_NR_RET_OP_CUT;
      A     "DOOR_EXTRACTOR_DB".DOOR_EXT_AUTO_SS;
      =     L 0.0;
      A     L 0.0;
      AN    "DOOR_EXTRACTOR_DB".SLEW_NR_AUTO_RET_OVR;
      A     "ONE_SECOND_PULSE";
      JNB   M014;
      L     1;
      L     "DOOR_EXTRACTOR_DB".SLEW_NR_ATO_RET_DL_T;
      +I;
      T     "DOOR_EXTRACTOR_DB".SLEW_NR_ATO_RET_DL_T;
M014: NOP   0;
      A     L 0.0;
      A(;
      L     "DOOR_EXTRACTOR_DB".SLEW_NR_ATO_RET_DL_T;
      L     "DOOR_EXTRACTOR_DB".SLEW_NR_AUTO_RET_DEL;
      >=I;
      );
      =     "DOOR_EXTRACTOR_DB".SLEW_NR_AUTO_RET_OVR;
NETWORK
TITLE =
      A     "ALWAYS_ON";
      A(;
      A(;
      O     "DOOR_EXTRACTOR_DB".SLEW_NOR_RET_COMMAND;
      O     "DOOR_EXTRACTOR_DB".SLEW_SLOW_RET_CMD;
      );
      A     "HALF_SECOND_PULSE_TRAIN";
      O     "DOOR_EXTRACTOR_DB".SLEW_NR_RET_OP_CUT;
      O     "MAIN_POWER_DB".LAMP_TEST_PB;
      );
      =     "DOOR_EXTRACTOR_DB".SLEW_RET_IND;
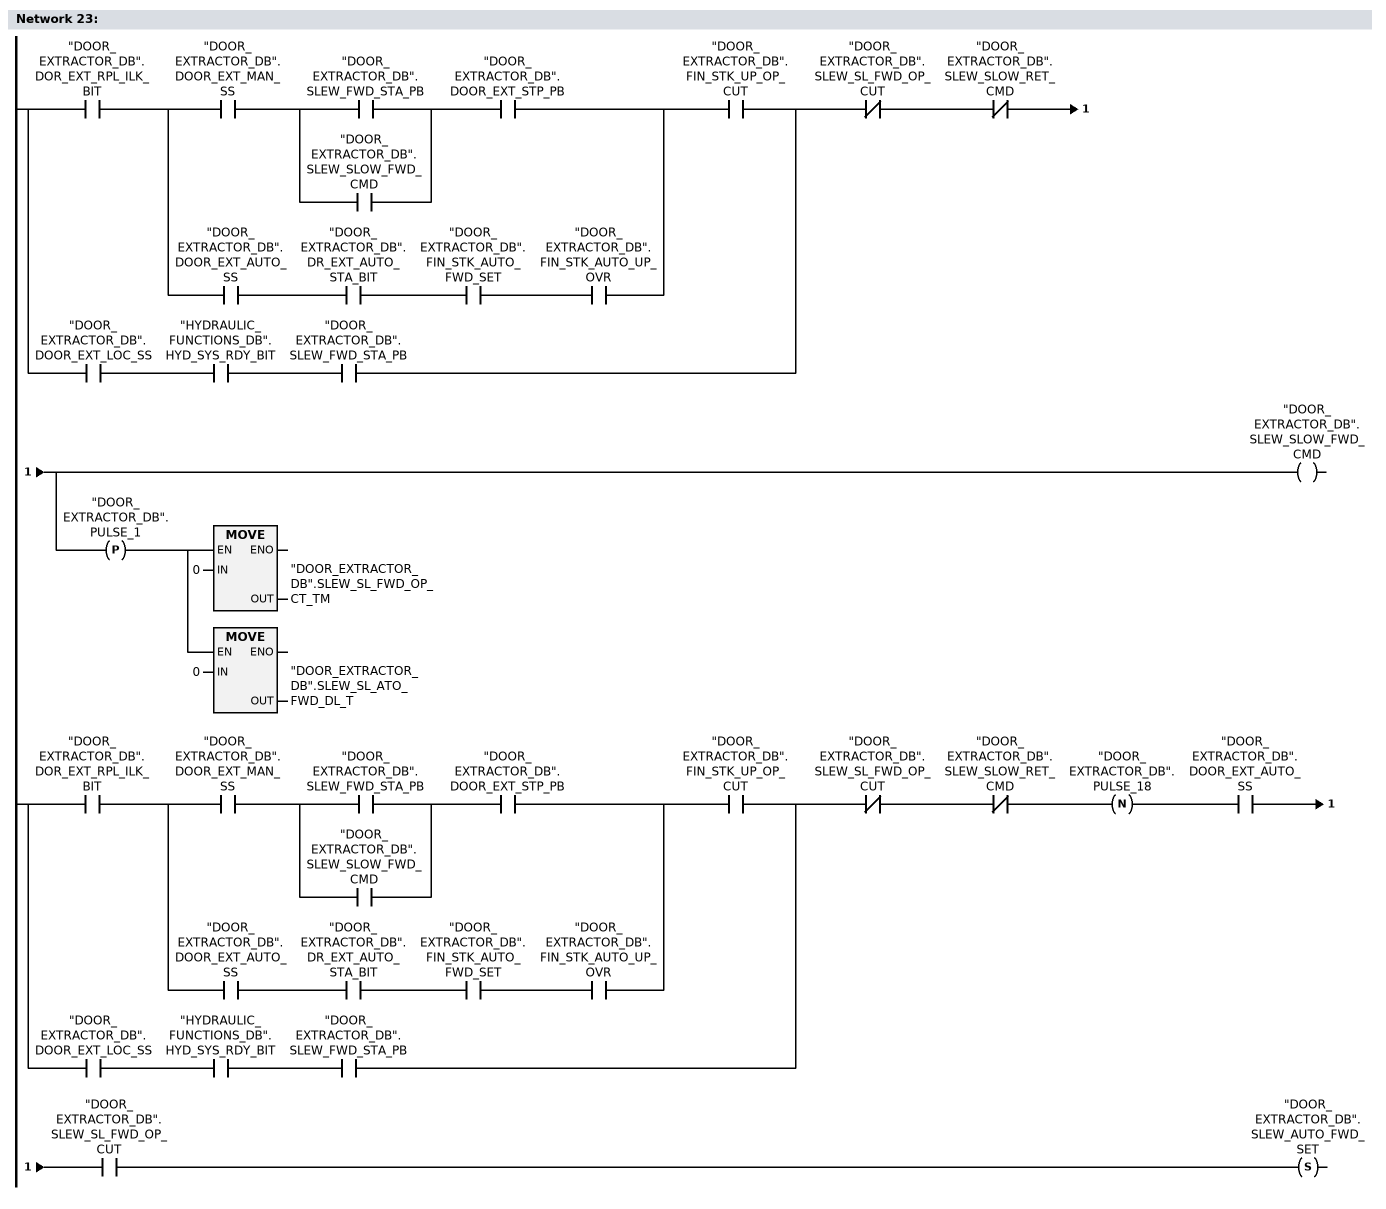
NETWORK
TITLE =
      A(;
      A     "DOOR_EXTRACTOR_DB".DOR_EXT_RPL_ILK_BIT;
      A(;
      A     "DOOR_EXTRACTOR_DB".DOOR_EXT_MAN_SS;
      A(;
      O     "DOOR_EXTRACTOR_DB".SLEW_FWD_STA_PB;
      O     "DOOR_EXTRACTOR_DB".SLEW_SLOW_FWD_CMD;
      );
      A     "DOOR_EXTRACTOR_DB".DOOR_EXT_STP_PB;
      O;
      A     "DOOR_EXTRACTOR_DB".DOOR_EXT_AUTO_SS;
      A     "DOOR_EXTRACTOR_DB".DR_EXT_AUTO_STA_BIT;
      A     "DOOR_EXTRACTOR_DB".FIN_STK_AUTO_FWD_SET;
      A     "DOOR_EXTRACTOR_DB".FIN_STK_AUTO_UP_OVR;
      );
      A     "DOOR_EXTRACTOR_DB".FIN_STK_UP_OP_CUT;
      O;
      A     "DOOR_EXTRACTOR_DB".DOOR_EXT_LOC_SS;
      A     "HYDRAULIC_FUNCTIONS_DB".HYD_SYS_RDY_BIT;
      A     "DOOR_EXTRACTOR_DB".SLEW_FWD_STA_PB;
      );
      AN    "DOOR_EXTRACTOR_DB".SLEW_SL_FWD_OP_CUT;
      AN    "DOOR_EXTRACTOR_DB".SLEW_SLOW_RET_CMD;
      =     L 0.0;
      A     L 0.0;
      BLD   102;
      =     "DOOR_EXTRACTOR_DB".SLEW_SLOW_FWD_CMD;
      A(;
      A     L 0.0;
      FN    "DOOR_EXTRACTOR_DB".PULSE_18;
      );
      A     "DOOR_EXTRACTOR_DB".DOOR_EXT_AUTO_SS;
      A     "DOOR_EXTRACTOR_DB".SLEW_SL_FWD_OP_CUT;
      S     "DOOR_EXTRACTOR_DB".SLEW_AUTO_FWD_SET;
      A     L 0.0;
      FP    "DOOR_EXTRACTOR_DB".PULSE_1;
      =     L 0.1;
      A     L 0.1;
      JNB   M015;
      L     0;
      T     "DOOR_EXTRACTOR_DB".SLEW_SL_FWD_OP_CT_TM;
M015: NOP   0;
      A     L 0.1;
      JNB   M016;
      L     0;
      T     "DOOR_EXTRACTOR_DB".SLEW_SL_ATO_FWD_DL_T;
M016: NOP   0;
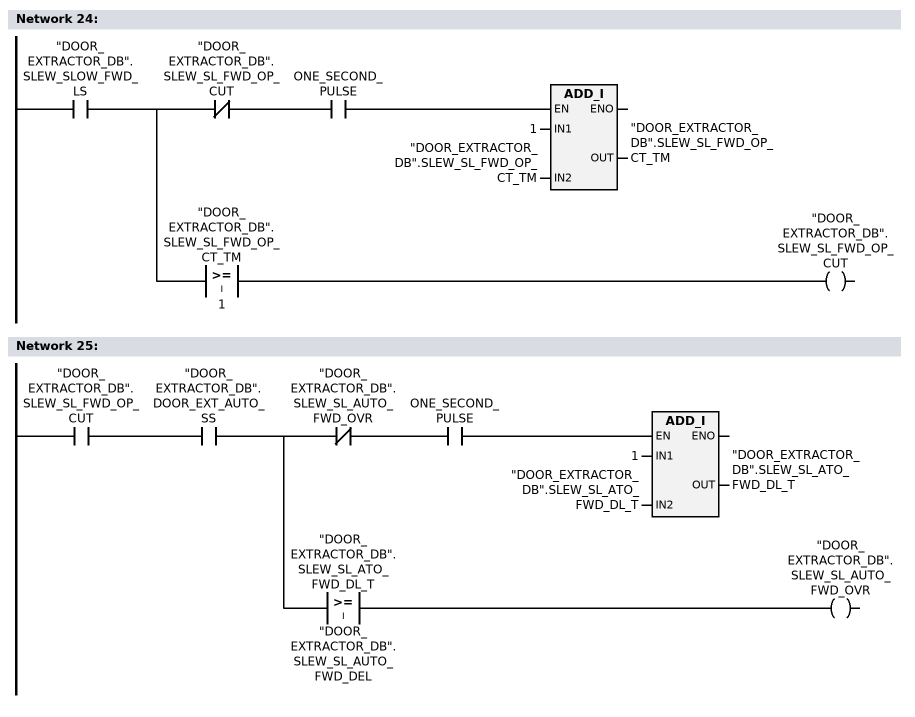
NETWORK
TITLE =
      A     "DOOR_EXTRACTOR_DB".SLEW_SLOW_FWD_LS;
      =     L 0.0;
      A     L 0.0;
      AN    "DOOR_EXTRACTOR_DB".SLEW_SL_FWD_OP_CUT;
      A     "ONE_SECOND_PULSE";
      JNB   M017;
      L     1;
      L     "DOOR_EXTRACTOR_DB".SLEW_SL_FWD_OP_CT_TM;
      +I;
      T     "DOOR_EXTRACTOR_DB".SLEW_SL_FWD_OP_CT_TM;
M017: NOP   0;
      A     L 0.0;
      A(;
      L     "DOOR_EXTRACTOR_DB".SLEW_SL_FWD_OP_CT_TM;
      L     1;
      >=I;
      );
      =     "DOOR_EXTRACTOR_DB".SLEW_SL_FWD_OP_CUT;
NETWORK
TITLE =
      A     "DOOR_EXTRACTOR_DB".SLEW_SL_FWD_OP_CUT;
      A     "DOOR_EXTRACTOR_DB".DOOR_EXT_AUTO_SS;
      =     L 0.0;
      A     L 0.0;
      AN    "DOOR_EXTRACTOR_DB".SLEW_SL_AUTO_FWD_OVR;
      A     "ONE_SECOND_PULSE";
      JNB   M018;
      L     1;
      L     "DOOR_EXTRACTOR_DB".SLEW_SL_ATO_FWD_DL_T;
      +I;
      T     "DOOR_EXTRACTOR_DB".SLEW_SL_ATO_FWD_DL_T;
M018: NOP   0;
      A     L 0.0;
      A(;
      L     "DOOR_EXTRACTOR_DB".SLEW_SL_ATO_FWD_DL_T;
      L     "DOOR_EXTRACTOR_DB".SLEW_SL_AUTO_FWD_DEL;
      >=I;
      );
      =     "DOOR_EXTRACTOR_DB".SLEW_SL_AUTO_FWD_OVR;
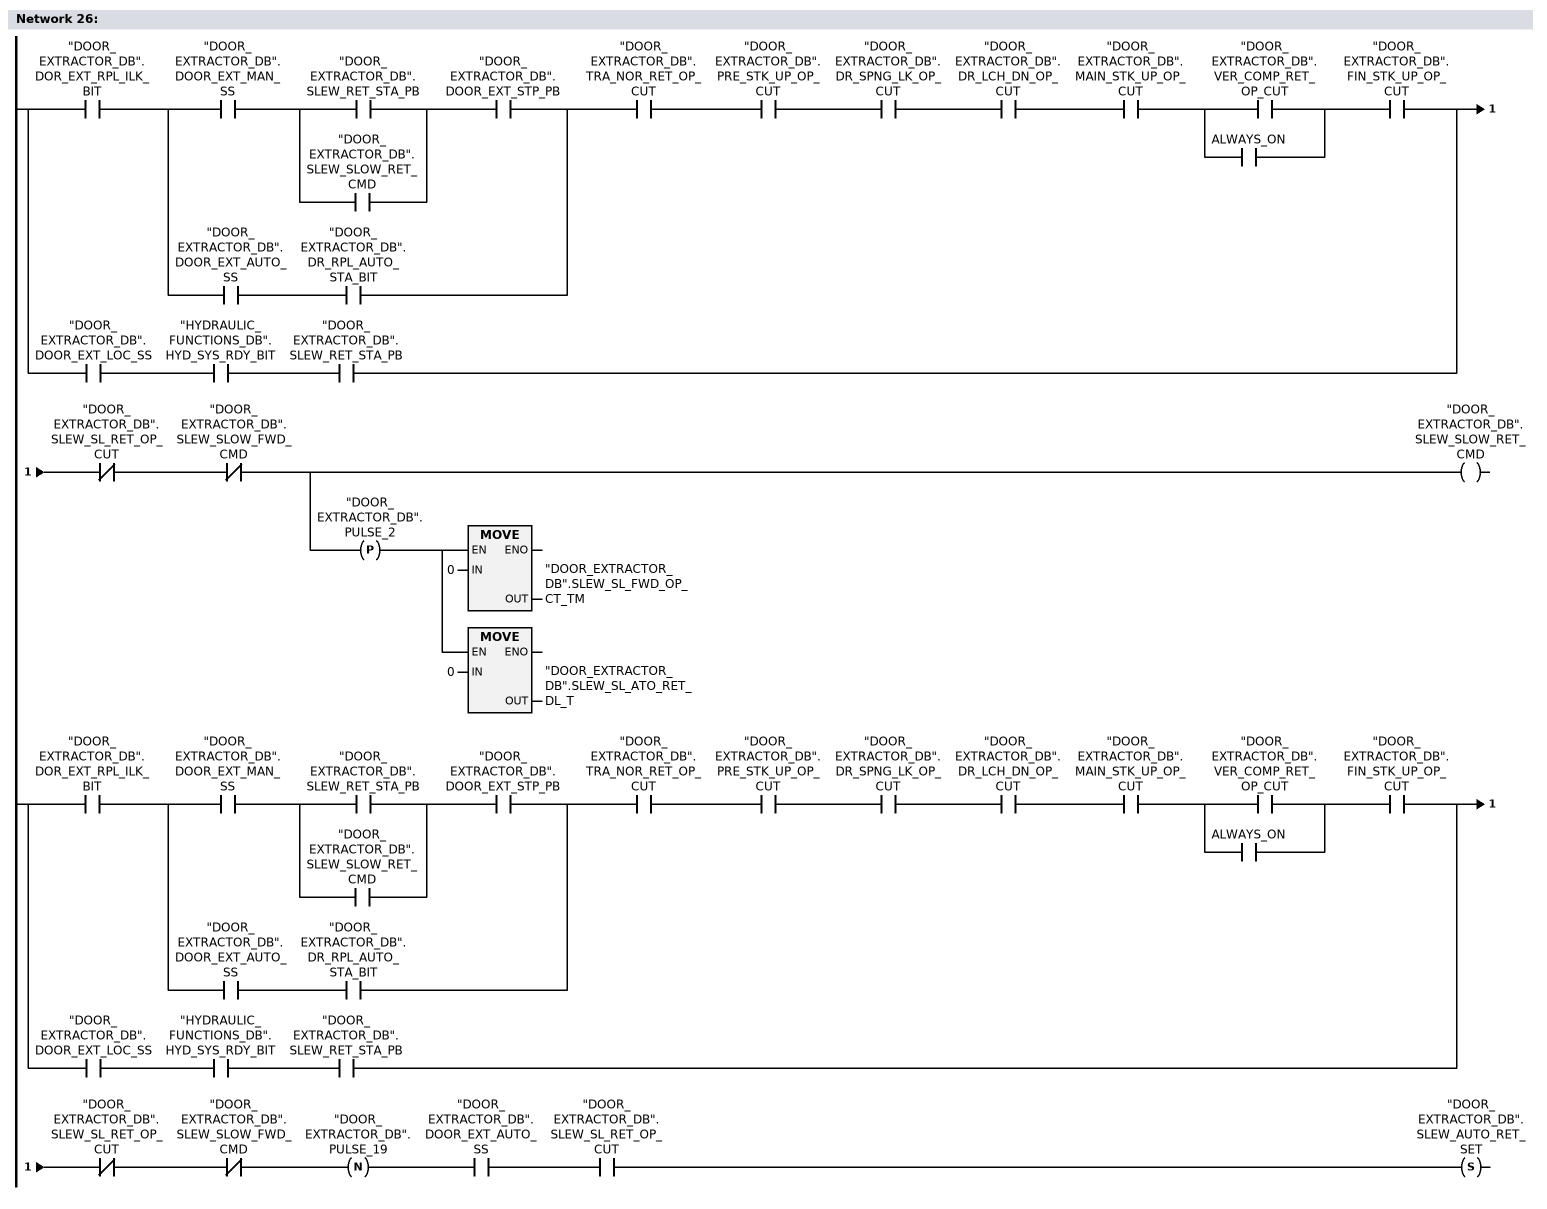
NETWORK
TITLE =
      A(;
      A     "DOOR_EXTRACTOR_DB".DOR_EXT_RPL_ILK_BIT;
      A(;
      A     "DOOR_EXTRACTOR_DB".DOOR_EXT_MAN_SS;
      A(;
      O     "DOOR_EXTRACTOR_DB".SLEW_RET_STA_PB;
      O     "DOOR_EXTRACTOR_DB".SLEW_SLOW_RET_CMD;
      );
      A     "DOOR_EXTRACTOR_DB".DOOR_EXT_STP_PB;
      O;
      A     "DOOR_EXTRACTOR_DB".DOOR_EXT_AUTO_SS;
      A     "DOOR_EXTRACTOR_DB".DR_RPL_AUTO_STA_BIT;
      );
      A     "DOOR_EXTRACTOR_DB".TRA_NOR_RET_OP_CUT;
      A     "DOOR_EXTRACTOR_DB".PRE_STK_UP_OP_CUT;
      A     "DOOR_EXTRACTOR_DB".DR_SPNG_LK_OP_CUT;
      A     "DOOR_EXTRACTOR_DB".DR_LCH_DN_OP_CUT;
      A     "DOOR_EXTRACTOR_DB".MAIN_STK_UP_OP_CUT;
      A(;
      O     "DOOR_EXTRACTOR_DB".VER_COMP_RET_OP_CUT;
      O     "ALWAYS_ON";
      );
      A     "DOOR_EXTRACTOR_DB".FIN_STK_UP_OP_CUT;
      O;
      A     "DOOR_EXTRACTOR_DB".DOOR_EXT_LOC_SS;
      A     "HYDRAULIC_FUNCTIONS_DB".HYD_SYS_RDY_BIT;
      A     "DOOR_EXTRACTOR_DB".SLEW_RET_STA_PB;
      );
      AN    "DOOR_EXTRACTOR_DB".SLEW_SL_RET_OP_CUT;
      AN    "DOOR_EXTRACTOR_DB".SLEW_SLOW_FWD_CMD;
      =     L 0.0;
      A     L 0.0;
      BLD   102;
      =     "DOOR_EXTRACTOR_DB".SLEW_SLOW_RET_CMD;
      A(;
      A     L 0.0;
      FN    "DOOR_EXTRACTOR_DB".PULSE_19;
      );
      A     "DOOR_EXTRACTOR_DB".DOOR_EXT_AUTO_SS;
      A     "DOOR_EXTRACTOR_DB".SLEW_SL_RET_OP_CUT;
      S     "DOOR_EXTRACTOR_DB".SLEW_AUTO_RET_SET;
      A     L 0.0;
      FP    "DOOR_EXTRACTOR_DB".PULSE_2;
      =     L 0.1;
      A     L 0.1;
      JNB   M019;
      L     0;
      T     "DOOR_EXTRACTOR_DB".SLEW_SL_FWD_OP_CT_TM;
M019: NOP   0;
      A     L 0.1;
      JNB   M020;
      L     0;
      T     "DOOR_EXTRACTOR_DB".SLEW_SL_ATO_RET_DL_T;
M020: NOP   0;
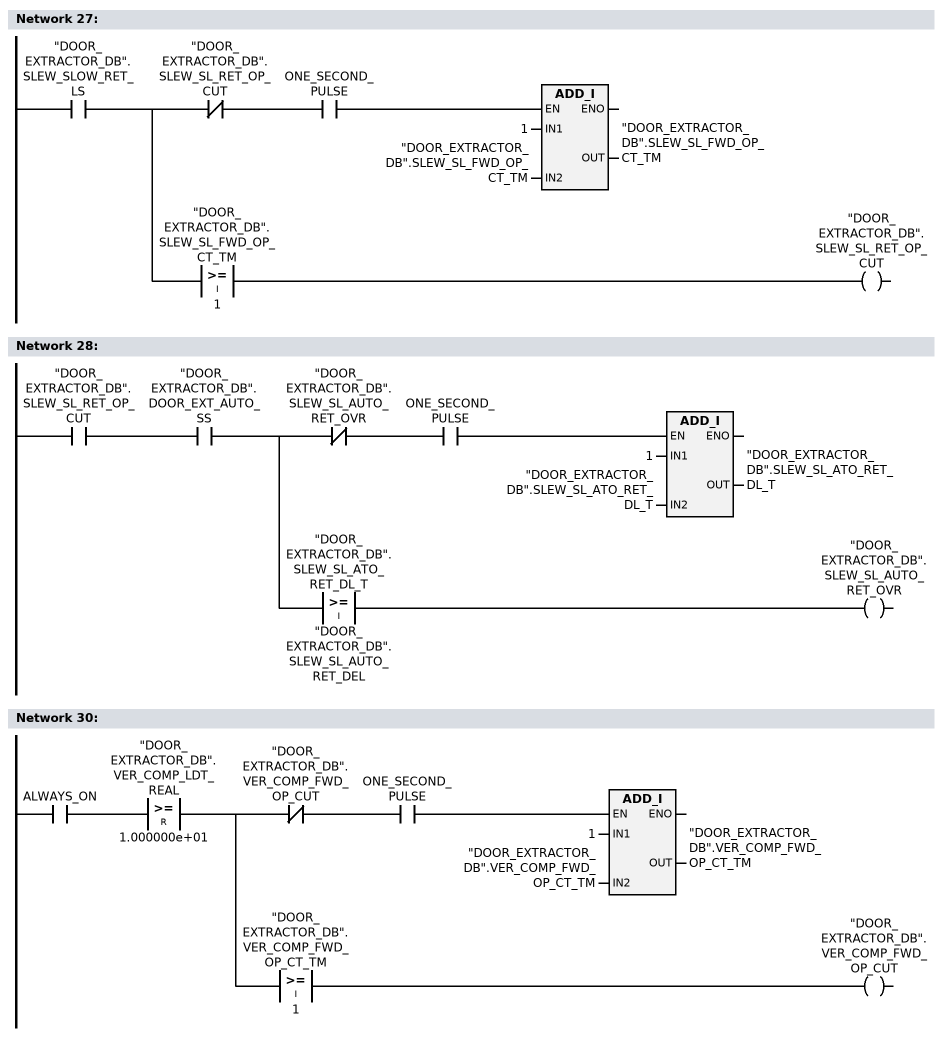
NETWORK
TITLE =
      A     "DOOR_EXTRACTOR_DB".SLEW_SLOW_RET_LS;
      =     L 0.0;
      A     L 0.0;
      AN    "DOOR_EXTRACTOR_DB".SLEW_SL_RET_OP_CUT;
      A     "ONE_SECOND_PULSE";
      JNB   M021;
      L     1;
      L     "DOOR_EXTRACTOR_DB".SLEW_SL_FWD_OP_CT_TM;
      +I;
      T     "DOOR_EXTRACTOR_DB".SLEW_SL_FWD_OP_CT_TM;
M021: NOP   0;
      A     L 0.0;
      A(;
      L     "DOOR_EXTRACTOR_DB".SLEW_SL_FWD_OP_CT_TM;
      L     1;
      >=I;
      );
      =     "DOOR_EXTRACTOR_DB".SLEW_SL_RET_OP_CUT;
NETWORK
TITLE =
      A     "DOOR_EXTRACTOR_DB".SLEW_SL_RET_OP_CUT;
      A     "DOOR_EXTRACTOR_DB".DOOR_EXT_AUTO_SS;
      =     L 0.0;
      A     L 0.0;
      AN    "DOOR_EXTRACTOR_DB".SLEW_SL_AUTO_RET_OVR;
      A     "ONE_SECOND_PULSE";
      JNB   M022;
      L     1;
      L     "DOOR_EXTRACTOR_DB".SLEW_SL_ATO_RET_DL_T;
      +I;
      T     "DOOR_EXTRACTOR_DB".SLEW_SL_ATO_RET_DL_T;
M022: NOP   0;
      A     L 0.0;
      A(;
      L     "DOOR_EXTRACTOR_DB".SLEW_SL_ATO_RET_DL_T;
      L     "DOOR_EXTRACTOR_DB".SLEW_SL_AUTO_RET_DEL;
      >=I;
      );
      =     "DOOR_EXTRACTOR_DB".SLEW_SL_AUTO_RET_OVR;
NETWORK
TITLE =
      A(;
      A     "DOOR_EXTRACTOR_DB".DOR_EXT_RPL_ILK_BIT;
      A(;
      A     "DOOR_EXTRACTOR_DB".DOOR_EXT_MAN_SS;
      A(;
      O     "DOOR_EXTRACTOR_DB".VER_COMP_FWD_STA_PB;
      O     "DOOR_EXTRACTOR_DB".VER_COMP_FWD_CMD;
      );
      A     "DOOR_EXTRACTOR_DB".DOOR_EXT_STP_PB;
      O;
      A     "DOOR_EXTRACTOR_DB".DOOR_EXT_AUTO_SS;
      A(;
      A     "DOOR_EXTRACTOR_DB".DR_EXT_AUTO_STA_BIT;
      A(;
      ON    "DOOR_EXTRACTOR_DB".VER_COMP_AUTO_FWD_SET;
      O     "ALWAYS_ON";
      );
      O;
      A     "DOOR_EXTRACTOR_DB".DR_RPL_AUTO_STA_BIT;
      A     "DOOR_EXTRACTOR_DB".FIN_STK_AUTO_RET_SET;
      A(;
      ON    "DOOR_EXTRACTOR_DB".VER_COMP_AUTO_FWD_SET;
      O     "ALWAYS_ON";
      );
      );
      );
      A(;
      A     "DOOR_EXTRACTOR_DB".SLEW_NR_RET_OP_CUT;
      A     "DOOR_EXTRACTOR_DB".PRE_STK_DN_OP_CUT;
      A     "DOOR_EXTRACTOR_DB".MAIN_STK_DN_OP_CUT;
      A     "DOOR_EXTRACTOR_DB".DR_LCH_UP_OP_CUT;
      A     "DOOR_EXTRACTOR_DB".DR_SPNG_UNLK_OP_CUT;
      O;
      A     "DOOR_EXTRACTOR_DB".SLEW_NR_RET_OP_CUT;
      A     "DOOR_EXTRACTOR_DB".TRA_NOR_RET_OP_CUT;
      A     "DOOR_EXTRACTOR_DB".PRE_STK_UP_OP_CUT;
      A     "DOOR_EXTRACTOR_DB".DR_SPNG_LK_OP_CUT;
      A     "DOOR_EXTRACTOR_DB".DR_LCH_DN_OP_CUT;
      A     "DOOR_EXTRACTOR_DB".MAIN_STK_UP_OP_CUT;
      A     "DOOR_EXTRACTOR_DB".FIN_STK_DN_OP_CUT;
      );
      O;
      A     "DOOR_EXTRACTOR_DB".DOOR_EXT_LOC_SS;
      A     "HYDRAULIC_FUNCTIONS_DB".HYD_SYS_RDY_BIT;
      A     "DOOR_EXTRACTOR_DB".VER_COMP_FWD_STA_PB;
      );
      A(;
      ON    "DOOR_EXTRACTOR_DB".VER_COMP_FWD_OP_CUT;
      O     "ALWAYS_ON";
      );
      AN    "DOOR_EXTRACTOR_DB".VER_COMP_RET_CMD;
      =     L 0.0;
      A     L 0.0;
      AN    "DOOR_EXTRACTOR_DB".DOOR_EXT_AUTO_SS;
      =     L 0.1;
      A     L 0.1;
      BLD   102;
      =     "DOOR_EXTRACTOR_DB".VER_COMP_FWD_CMD;
      A(;
      A     L 0.1;
      FN    "DOOR_EXTRACTOR_DB".PULSE_20;
      );
      A     "DOOR_EXTRACTOR_DB".VER_COMP_FWD_OP_CUT;
      A     "DOOR_EXTRACTOR_DB".DOOR_EXT_AUTO_SS;
      S     "DOOR_EXTRACTOR_DB".VER_COMP_AUTO_FWD_SET;
      A     L 0.0;
      FP    "DOOR_EXTRACTOR_DB".PULSE_3;
      =     L 0.1;
      A     L 0.1;
      A     "DOOR_EXTRACTOR_DB".DOOR_EXT_AUTO_SS;
      S     "DOOR_EXTRACTOR_DB".VER_COMP_AUTO_FWD_SET;
      A     L 0.1;
      JNB   M023;
      L     0;
      T     "DOOR_EXTRACTOR_DB".VER_COMP_FWD_OP_CT_TM;
M023: NOP   0;
      A     L 0.1;
      JNB   M024;
      L     0;
      T     "DOOR_EXTRACTOR_DB".VER_COMP_ATO_FWD_DL_T;
M024: NOP   0;
NETWORK
TITLE =
      A     "ALWAYS_ON";
      A(;
      L     "DOOR_EXTRACTOR_DB".VER_COMP_LDT_REAL;
      L     1.000000e+01;
      >=R;
      );
      =     L 0.0;
      A     L 0.0;
      AN    "DOOR_EXTRACTOR_DB".VER_COMP_FWD_OP_CUT;
      A     "ONE_SECOND_PULSE";
      JNB   M025;
      L     1;
      L     "DOOR_EXTRACTOR_DB".VER_COMP_FWD_OP_CT_TM;
      +I;
      T     "DOOR_EXTRACTOR_DB".VER_COMP_FWD_OP_CT_TM;
M025: NOP   0;
      A     L 0.0;
      A(;
      L     "DOOR_EXTRACTOR_DB".VER_COMP_FWD_OP_CT_TM;
      L     1;
      >=I;
      );
      =     "DOOR_EXTRACTOR_DB".VER_COMP_FWD_OP_CUT;
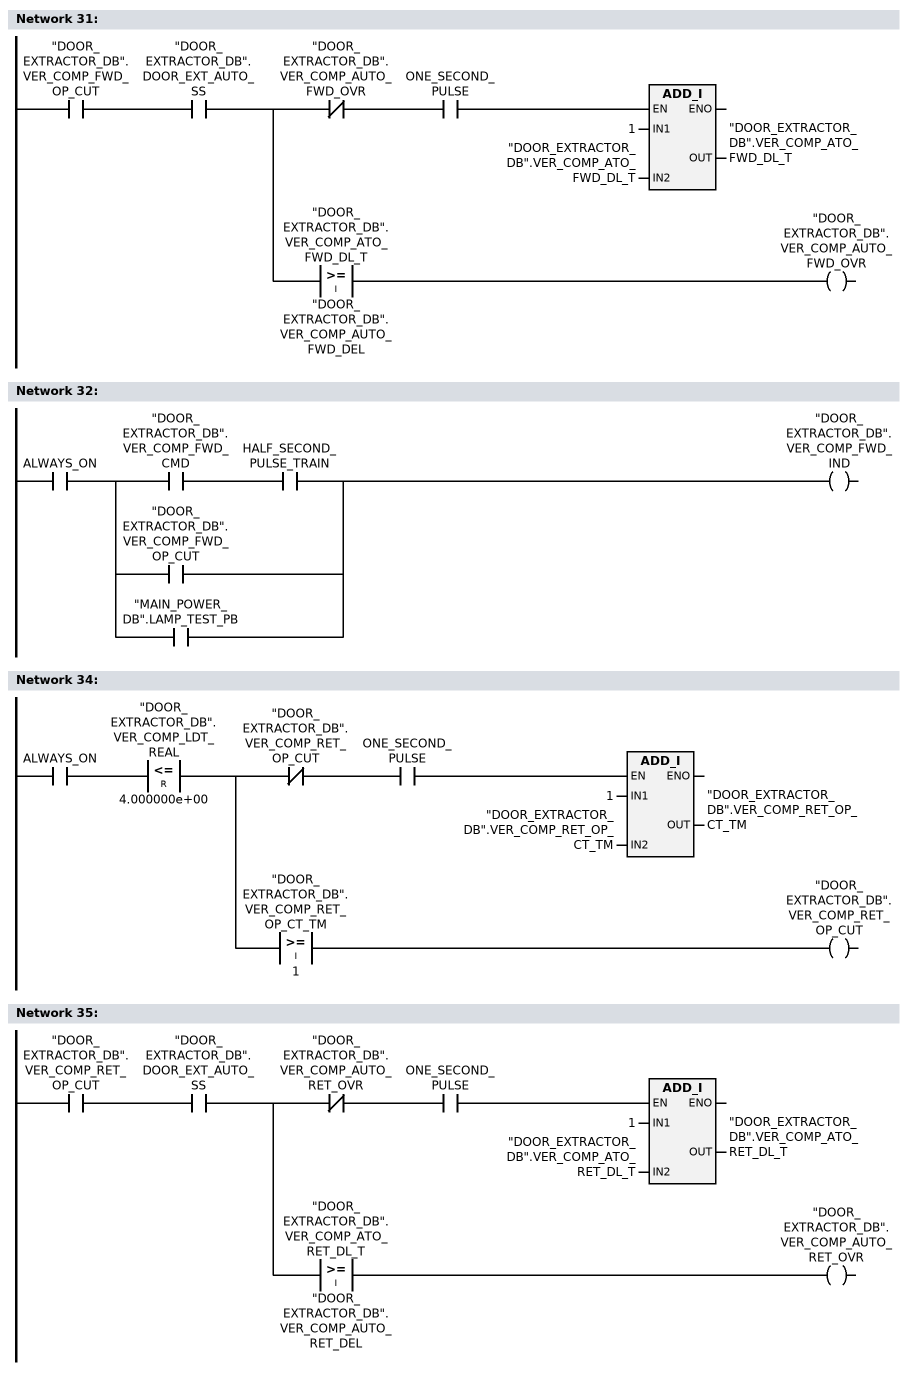
NETWORK
TITLE =
      A     "DOOR_EXTRACTOR_DB".VER_COMP_FWD_OP_CUT;
      A     "DOOR_EXTRACTOR_DB".DOOR_EXT_AUTO_SS;
      =     L 0.0;
      A     L 0.0;
      AN    "DOOR_EXTRACTOR_DB".VER_COMP_AUTO_FWD_OVR;
      A     "ONE_SECOND_PULSE";
      JNB   M026;
      L     1;
      L     "DOOR_EXTRACTOR_DB".VER_COMP_ATO_FWD_DL_T;
      +I;
      T     "DOOR_EXTRACTOR_DB".VER_COMP_ATO_FWD_DL_T;
M026: NOP   0;
      A     L 0.0;
      A(;
      L     "DOOR_EXTRACTOR_DB".VER_COMP_ATO_FWD_DL_T;
      L     "DOOR_EXTRACTOR_DB".VER_COMP_AUTO_FWD_DEL;
      >=I;
      );
      =     "DOOR_EXTRACTOR_DB".VER_COMP_AUTO_FWD_OVR;
NETWORK
TITLE =
      A     "ALWAYS_ON";
      A(;
      A     "DOOR_EXTRACTOR_DB".VER_COMP_FWD_CMD;
      A     "HALF_SECOND_PULSE_TRAIN";
      O     "DOOR_EXTRACTOR_DB".VER_COMP_FWD_OP_CUT;
      O     "MAIN_POWER_DB".LAMP_TEST_PB;
      );
      =     "DOOR_EXTRACTOR_DB".VER_COMP_FWD_IND;
NETWORK
TITLE =
      A(;
      A     "DOOR_EXTRACTOR_DB".DOR_EXT_RPL_ILK_BIT;
      A(;
      A     "DOOR_EXTRACTOR_DB".DOOR_EXT_MAN_SS;
      A(;
      O     "DOOR_EXTRACTOR_DB".VER_COMP_RET_STA_PB;
      O     "DOOR_EXTRACTOR_DB".VER_COMP_RET_CMD;
      );
      A     "DOOR_EXTRACTOR_DB".DOOR_EXT_STP_PB;
      O;
      A     "DOOR_EXTRACTOR_DB".DOOR_EXT_AUTO_SS;
      A(;
      A     "DOOR_EXTRACTOR_DB".DR_EXT_AUTO_STA_BIT;
      A     "DOOR_EXTRACTOR_DB".TRA_AUTO_RET_SET;
      A     "DOOR_EXTRACTOR_DB".TRA_NOR_AUTO_RET_OVR;
      O;
      A     "DOOR_EXTRACTOR_DB".DR_RPL_AUTO_STA_BIT;
      A     "DOOR_EXTRACTOR_DB".TRA_AUTO_RET_SET;
      A     "DOOR_EXTRACTOR_DB".TRA_NOR_AUTO_RET_OVR;
      );
      );
      A(;
      A     "DOOR_EXTRACTOR_DB".SLEW_NR_RET_OP_CUT;
      A     "DOOR_EXTRACTOR_DB".TRA_NOR_RET_OP_CUT;
      A     "DOOR_EXTRACTOR_DB".PRE_STK_UP_OP_CUT;
      A     "DOOR_EXTRACTOR_DB".DR_SPNG_LK_OP_CUT;
      A     "DOOR_EXTRACTOR_DB".DR_LCH_DN_OP_CUT;
      A     "DOOR_EXTRACTOR_DB".MAIN_STK_UP_OP_CUT;
      O;
      A     "DOOR_EXTRACTOR_DB".SLEW_NR_RET_OP_CUT;
      A     "DOOR_EXTRACTOR_DB".TRA_NOR_RET_OP_CUT;
      A     "DOOR_EXTRACTOR_DB".PRE_STK_DN_OP_CUT;
      A     "DOOR_EXTRACTOR_DB".DR_SPNG_UNLK_OP_CUT;
      A     "DOOR_EXTRACTOR_DB".DR_LCH_UP_OP_CUT;
      A     "DOOR_EXTRACTOR_DB".MAIN_STK_DN_OP_CUT;
      A     "DOOR_EXTRACTOR_DB".FIN_STK_DN_OP_CUT;
      );
      O;
      A     "DOOR_EXTRACTOR_DB".DOOR_EXT_LOC_SS;
      A     "HYDRAULIC_FUNCTIONS_DB".HYD_SYS_RDY_BIT;
      A     "DOOR_EXTRACTOR_DB".VER_COMP_RET_STA_PB;
      );
      A(;
      ON    "DOOR_EXTRACTOR_DB".VER_COMP_RET_OP_CUT;
      O     "ALWAYS_ON";
      );
      AN    "DOOR_EXTRACTOR_DB".VER_COMP_FWD_CMD;
      =     L 0.0;
      A     L 0.0;
      AN    "DOOR_EXTRACTOR_DB".DOOR_EXT_AUTO_SS;
      =     L 0.1;
      A     L 0.1;
      BLD   102;
      =     "DOOR_EXTRACTOR_DB".VER_COMP_RET_CMD;
      A(;
      A     L 0.1;
      FN    "DOOR_EXTRACTOR_DB".PULSE_21;
      );
      A     "DOOR_EXTRACTOR_DB".DOOR_EXT_AUTO_SS;
      A     "DOOR_EXTRACTOR_DB".VER_COMP_RET_OP_CUT;
      S     "DOOR_EXTRACTOR_DB".VER_COMP_AUTO_RET_SET;
      A     L 0.0;
      FP    "DOOR_EXTRACTOR_DB".PULSE_4;
      =     L 0.1;
      A     L 0.1;
      A     "DOOR_EXTRACTOR_DB".DOOR_EXT_AUTO_SS;
      S     "DOOR_EXTRACTOR_DB".VER_COMP_AUTO_RET_SET;
      A     L 0.1;
      JNB   M027;
      L     0;
      T     "DOOR_EXTRACTOR_DB".VER_COMP_RET_OP_CT_TM;
M027: NOP   0;
      A     L 0.1;
      JNB   M028;
      L     0;
      T     "DOOR_EXTRACTOR_DB".VER_COMP_ATO_RET_DL_T;
M028: NOP   0;
NETWORK
TITLE =
      A     "ALWAYS_ON";
      A(;
      L     "DOOR_EXTRACTOR_DB".VER_COMP_LDT_REAL;
      L     4.000000e+00;
      <=R;
      );
      =     L 0.0;
      A     L 0.0;
      AN    "DOOR_EXTRACTOR_DB".VER_COMP_RET_OP_CUT;
      A     "ONE_SECOND_PULSE";
      JNB   M029;
      L     1;
      L     "DOOR_EXTRACTOR_DB".VER_COMP_RET_OP_CT_TM;
      +I;
      T     "DOOR_EXTRACTOR_DB".VER_COMP_RET_OP_CT_TM;
M029: NOP   0;
      A     L 0.0;
      A(;
      L     "DOOR_EXTRACTOR_DB".VER_COMP_RET_OP_CT_TM;
      L     1;
      >=I;
      );
      =     "DOOR_EXTRACTOR_DB".VER_COMP_RET_OP_CUT;
NETWORK
TITLE =
      A     "DOOR_EXTRACTOR_DB".VER_COMP_RET_OP_CUT;
      A     "DOOR_EXTRACTOR_DB".DOOR_EXT_AUTO_SS;
      =     L 0.0;
      A     L 0.0;
      AN    "DOOR_EXTRACTOR_DB".VER_COMP_AUTO_RET_OVR;
      A     "ONE_SECOND_PULSE";
      JNB   M030;
      L     1;
      L     "DOOR_EXTRACTOR_DB".VER_COMP_ATO_RET_DL_T;
      +I;
      T     "DOOR_EXTRACTOR_DB".VER_COMP_ATO_RET_DL_T;
M030: NOP   0;
      A     L 0.0;
      A(;
      L     "DOOR_EXTRACTOR_DB".VER_COMP_ATO_RET_DL_T;
      L     "DOOR_EXTRACTOR_DB".VER_COMP_AUTO_RET_DEL;
      >=I;
      );
      =     "DOOR_EXTRACTOR_DB".VER_COMP_AUTO_RET_OVR;
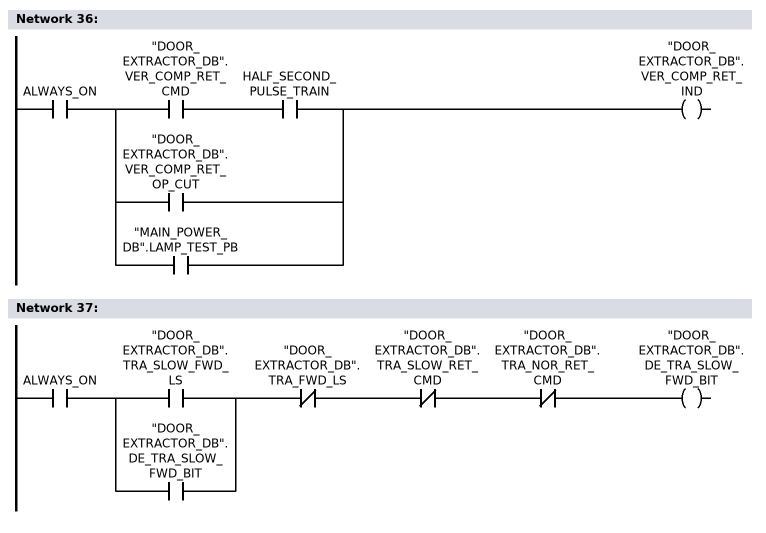
NETWORK
TITLE =
      A     "ALWAYS_ON";
      A(;
      A     "DOOR_EXTRACTOR_DB".VER_COMP_RET_CMD;
      A     "HALF_SECOND_PULSE_TRAIN";
      O     "DOOR_EXTRACTOR_DB".VER_COMP_RET_OP_CUT;
      O     "MAIN_POWER_DB".LAMP_TEST_PB;
      );
      =     "DOOR_EXTRACTOR_DB".VER_COMP_RET_IND;
NETWORK
TITLE =
      A     "ALWAYS_ON";
      A(;
      O     "DOOR_EXTRACTOR_DB".TRA_SLOW_FWD_LS;
      O     "DOOR_EXTRACTOR_DB".DE_TRA_SLOW_FWD_BIT;
      );
      AN    "DOOR_EXTRACTOR_DB".TRA_FWD_LS;
      AN    "DOOR_EXTRACTOR_DB".TRA_SLOW_RET_CMD;
      AN    "DOOR_EXTRACTOR_DB".TRA_NOR_RET_CMD;
      =     "DOOR_EXTRACTOR_DB".DE_TRA_SLOW_FWD_BIT;
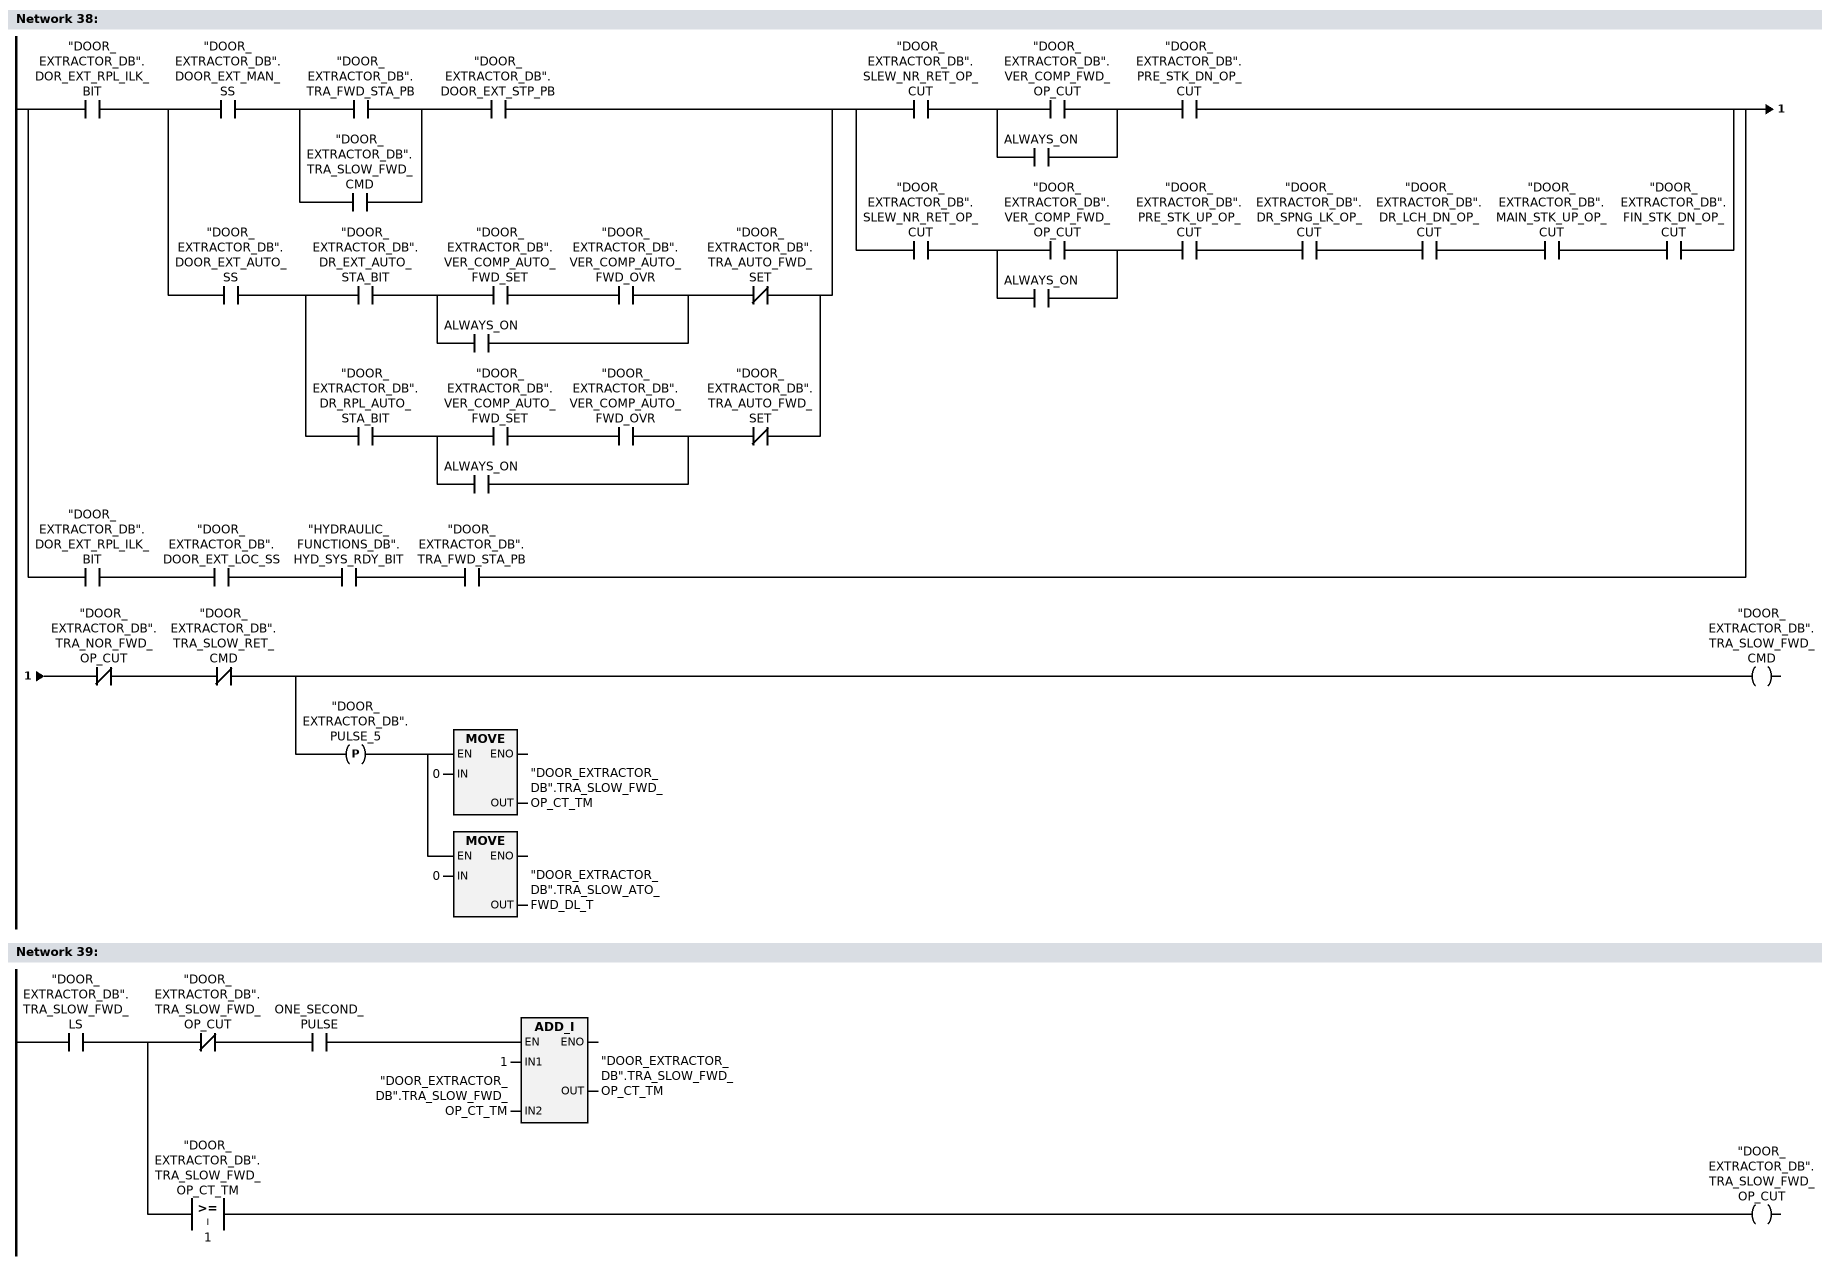
NETWORK
TITLE =
      A(;
      A     "DOOR_EXTRACTOR_DB".DOR_EXT_RPL_ILK_BIT;
      A(;
      A     "DOOR_EXTRACTOR_DB".DOOR_EXT_MAN_SS;
      A(;
      O     "DOOR_EXTRACTOR_DB".TRA_FWD_STA_PB;
      O     "DOOR_EXTRACTOR_DB".TRA_SLOW_FWD_CMD;
      );
      A     "DOOR_EXTRACTOR_DB".DOOR_EXT_STP_PB;
      O;
      A     "DOOR_EXTRACTOR_DB".DOOR_EXT_AUTO_SS;
      A(;
      A     "DOOR_EXTRACTOR_DB".DR_EXT_AUTO_STA_BIT;
      A(;
      A     "DOOR_EXTRACTOR_DB".VER_COMP_AUTO_FWD_SET;
      A     "DOOR_EXTRACTOR_DB".VER_COMP_AUTO_FWD_OVR;
      O     "ALWAYS_ON";
      );
      AN    "DOOR_EXTRACTOR_DB".TRA_AUTO_FWD_SET;
      O;
      A     "DOOR_EXTRACTOR_DB".DR_RPL_AUTO_STA_BIT;
      A(;
      A     "DOOR_EXTRACTOR_DB".VER_COMP_AUTO_FWD_SET;
      A     "DOOR_EXTRACTOR_DB".VER_COMP_AUTO_FWD_OVR;
      O     "ALWAYS_ON";
      );
      AN    "DOOR_EXTRACTOR_DB".TRA_AUTO_FWD_SET;
      );
      );
      A(;
      A     "DOOR_EXTRACTOR_DB".SLEW_NR_RET_OP_CUT;
      A(;
      O     "DOOR_EXTRACTOR_DB".VER_COMP_FWD_OP_CUT;
      O     "ALWAYS_ON";
      );
      A     "DOOR_EXTRACTOR_DB".PRE_STK_DN_OP_CUT;
      O;
      A     "DOOR_EXTRACTOR_DB".SLEW_NR_RET_OP_CUT;
      A(;
      O     "DOOR_EXTRACTOR_DB".VER_COMP_FWD_OP_CUT;
      O     "ALWAYS_ON";
      );
      A     "DOOR_EXTRACTOR_DB".PRE_STK_UP_OP_CUT;
      A     "DOOR_EXTRACTOR_DB".DR_SPNG_LK_OP_CUT;
      A     "DOOR_EXTRACTOR_DB".DR_LCH_DN_OP_CUT;
      A     "DOOR_EXTRACTOR_DB".MAIN_STK_UP_OP_CUT;
      A     "DOOR_EXTRACTOR_DB".FIN_STK_DN_OP_CUT;
      );
      O;
      A     "DOOR_EXTRACTOR_DB".DOR_EXT_RPL_ILK_BIT;
      A     "DOOR_EXTRACTOR_DB".DOOR_EXT_LOC_SS;
      A     "HYDRAULIC_FUNCTIONS_DB".HYD_SYS_RDY_BIT;
      A     "DOOR_EXTRACTOR_DB".TRA_FWD_STA_PB;
      );
      AN    "DOOR_EXTRACTOR_DB".TRA_NOR_FWD_OP_CUT;
      AN    "DOOR_EXTRACTOR_DB".TRA_SLOW_RET_CMD;
      =     L 0.0;
      A     L 0.0;
      BLD   102;
      =     "DOOR_EXTRACTOR_DB".TRA_SLOW_FWD_CMD;
      A     L 0.0;
      FP    "DOOR_EXTRACTOR_DB".PULSE_5;
      =     L 0.1;
      A     L 0.1;
      JNB   M031;
      L     0;
      T     "DOOR_EXTRACTOR_DB".TRA_SLOW_FWD_OP_CT_TM;
M031: NOP   0;
      A     L 0.1;
      JNB   M032;
      L     0;
      T     "DOOR_EXTRACTOR_DB".TRA_SLOW_ATO_FWD_DL_T;
M032: NOP   0;
NETWORK
TITLE =
      A     "DOOR_EXTRACTOR_DB".TRA_SLOW_FWD_LS;
      =     L 0.0;
      A     L 0.0;
      AN    "DOOR_EXTRACTOR_DB".TRA_SLOW_FWD_OP_CUT;
      A     "ONE_SECOND_PULSE";
      JNB   M033;
      L     1;
      L     "DOOR_EXTRACTOR_DB".TRA_SLOW_FWD_OP_CT_TM;
      +I;
      T     "DOOR_EXTRACTOR_DB".TRA_SLOW_FWD_OP_CT_TM;
M033: NOP   0;
      A     L 0.0;
      A(;
      L     "DOOR_EXTRACTOR_DB".TRA_SLOW_FWD_OP_CT_TM;
      L     1;
      >=I;
      );
      =     "DOOR_EXTRACTOR_DB".TRA_SLOW_FWD_OP_CUT;
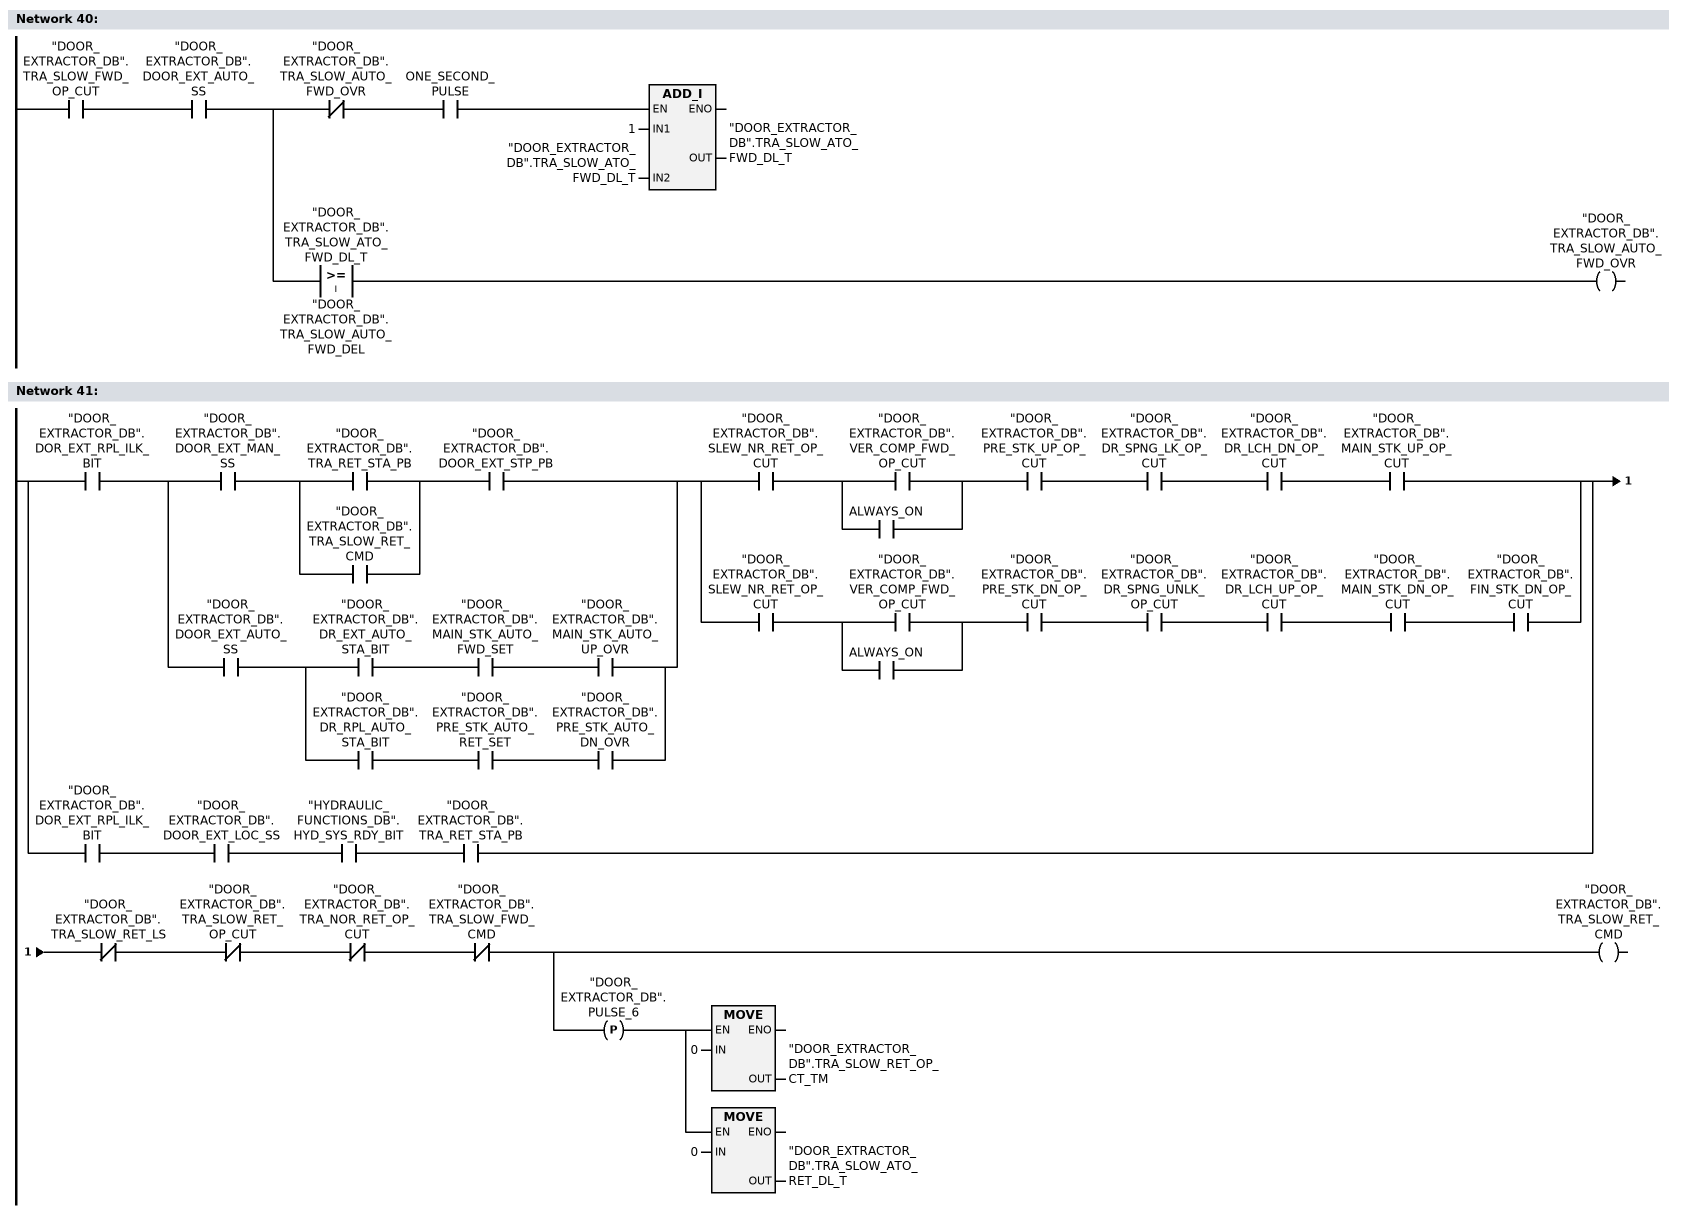
NETWORK
TITLE =
      A     "DOOR_EXTRACTOR_DB".TRA_SLOW_FWD_OP_CUT;
      A     "DOOR_EXTRACTOR_DB".DOOR_EXT_AUTO_SS;
      =     L 0.0;
      A     L 0.0;
      AN    "DOOR_EXTRACTOR_DB".TRA_SLOW_AUTO_FWD_OVR;
      A     "ONE_SECOND_PULSE";
      JNB   M034;
      L     1;
      L     "DOOR_EXTRACTOR_DB".TRA_SLOW_ATO_FWD_DL_T;
      +I;
      T     "DOOR_EXTRACTOR_DB".TRA_SLOW_ATO_FWD_DL_T;
M034: NOP   0;
      A     L 0.0;
      A(;
      L     "DOOR_EXTRACTOR_DB".TRA_SLOW_ATO_FWD_DL_T;
      L     "DOOR_EXTRACTOR_DB".TRA_SLOW_AUTO_FWD_DEL;
      >=I;
      );
      =     "DOOR_EXTRACTOR_DB".TRA_SLOW_AUTO_FWD_OVR;
NETWORK
TITLE =
      A(;
      A     "DOOR_EXTRACTOR_DB".DOR_EXT_RPL_ILK_BIT;
      A(;
      A     "DOOR_EXTRACTOR_DB".DOOR_EXT_MAN_SS;
      A(;
      O     "DOOR_EXTRACTOR_DB".TRA_RET_STA_PB;
      O     "DOOR_EXTRACTOR_DB".TRA_SLOW_RET_CMD;
      );
      A     "DOOR_EXTRACTOR_DB".DOOR_EXT_STP_PB;
      O;
      A     "DOOR_EXTRACTOR_DB".DOOR_EXT_AUTO_SS;
      A(;
      A     "DOOR_EXTRACTOR_DB".DR_EXT_AUTO_STA_BIT;
      A     "DOOR_EXTRACTOR_DB".MAIN_STK_AUTO_FWD_SET;
      A     "DOOR_EXTRACTOR_DB".MAIN_STK_AUTO_UP_OVR;
      O;
      A     "DOOR_EXTRACTOR_DB".DR_RPL_AUTO_STA_BIT;
      A     "DOOR_EXTRACTOR_DB".PRE_STK_AUTO_RET_SET;
      A     "DOOR_EXTRACTOR_DB".PRE_STK_AUTO_DN_OVR;
      );
      );
      A(;
      A     "DOOR_EXTRACTOR_DB".SLEW_NR_RET_OP_CUT;
      A(;
      O     "DOOR_EXTRACTOR_DB".VER_COMP_FWD_OP_CUT;
      O     "ALWAYS_ON";
      );
      A     "DOOR_EXTRACTOR_DB".PRE_STK_UP_OP_CUT;
      A     "DOOR_EXTRACTOR_DB".DR_SPNG_LK_OP_CUT;
      A     "DOOR_EXTRACTOR_DB".DR_LCH_DN_OP_CUT;
      A     "DOOR_EXTRACTOR_DB".MAIN_STK_UP_OP_CUT;
      O;
      A     "DOOR_EXTRACTOR_DB".SLEW_NR_RET_OP_CUT;
      A(;
      O     "DOOR_EXTRACTOR_DB".VER_COMP_FWD_OP_CUT;
      O     "ALWAYS_ON";
      );
      A     "DOOR_EXTRACTOR_DB".PRE_STK_DN_OP_CUT;
      A     "DOOR_EXTRACTOR_DB".DR_SPNG_UNLK_OP_CUT;
      A     "DOOR_EXTRACTOR_DB".DR_LCH_UP_OP_CUT;
      A     "DOOR_EXTRACTOR_DB".MAIN_STK_DN_OP_CUT;
      A     "DOOR_EXTRACTOR_DB".FIN_STK_DN_OP_CUT;
      );
      O;
      A     "DOOR_EXTRACTOR_DB".DOR_EXT_RPL_ILK_BIT;
      A     "DOOR_EXTRACTOR_DB".DOOR_EXT_LOC_SS;
      A     "HYDRAULIC_FUNCTIONS_DB".HYD_SYS_RDY_BIT;
      A     "DOOR_EXTRACTOR_DB".TRA_RET_STA_PB;
      );
      AN    "DOOR_EXTRACTOR_DB".TRA_SLOW_RET_LS;
      AN    "DOOR_EXTRACTOR_DB".TRA_SLOW_RET_OP_CUT;
      AN    "DOOR_EXTRACTOR_DB".TRA_NOR_RET_OP_CUT;
      AN    "DOOR_EXTRACTOR_DB".TRA_SLOW_FWD_CMD;
      =     L 0.0;
      A     L 0.0;
      BLD   102;
      =     "DOOR_EXTRACTOR_DB".TRA_SLOW_RET_CMD;
      A     L 0.0;
      FP    "DOOR_EXTRACTOR_DB".PULSE_6;
      =     L 0.1;
      A     L 0.1;
      JNB   M035;
      L     0;
      T     "DOOR_EXTRACTOR_DB".TRA_SLOW_RET_OP_CT_TM;
M035: NOP   0;
      A     L 0.1;
      JNB   M036;
      L     0;
      T     "DOOR_EXTRACTOR_DB".TRA_SLOW_ATO_RET_DL_T;
M036: NOP   0;
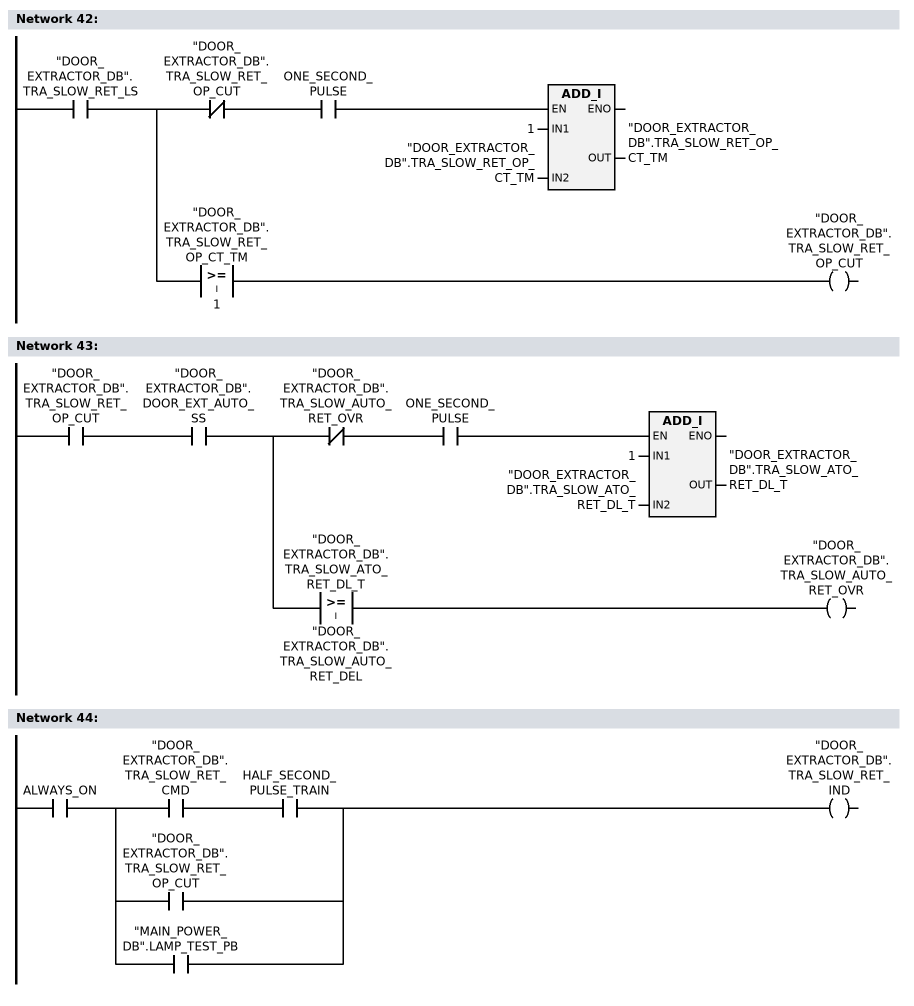
NETWORK
TITLE =
      A     "DOOR_EXTRACTOR_DB".TRA_SLOW_RET_LS;
      =     L 0.0;
      A     L 0.0;
      AN    "DOOR_EXTRACTOR_DB".TRA_SLOW_RET_OP_CUT;
      A     "ONE_SECOND_PULSE";
      JNB   M037;
      L     1;
      L     "DOOR_EXTRACTOR_DB".TRA_SLOW_RET_OP_CT_TM;
      +I;
      T     "DOOR_EXTRACTOR_DB".TRA_SLOW_RET_OP_CT_TM;
M037: NOP   0;
      A     L 0.0;
      A(;
      L     "DOOR_EXTRACTOR_DB".TRA_SLOW_RET_OP_CT_TM;
      L     1;
      >=I;
      );
      =     "DOOR_EXTRACTOR_DB".TRA_SLOW_RET_OP_CUT;
NETWORK
TITLE =
      A     "DOOR_EXTRACTOR_DB".TRA_SLOW_RET_OP_CUT;
      A     "DOOR_EXTRACTOR_DB".DOOR_EXT_AUTO_SS;
      =     L 0.0;
      A     L 0.0;
      AN    "DOOR_EXTRACTOR_DB".TRA_SLOW_AUTO_RET_OVR;
      A     "ONE_SECOND_PULSE";
      JNB   M038;
      L     1;
      L     "DOOR_EXTRACTOR_DB".TRA_SLOW_ATO_RET_DL_T;
      +I;
      T     "DOOR_EXTRACTOR_DB".TRA_SLOW_ATO_RET_DL_T;
M038: NOP   0;
      A     L 0.0;
      A(;
      L     "DOOR_EXTRACTOR_DB".TRA_SLOW_ATO_RET_DL_T;
      L     "DOOR_EXTRACTOR_DB".TRA_SLOW_AUTO_RET_DEL;
      >=I;
      );
      =     "DOOR_EXTRACTOR_DB".TRA_SLOW_AUTO_RET_OVR;
NETWORK
TITLE =
      A     "ALWAYS_ON";
      A(;
      A     "DOOR_EXTRACTOR_DB".TRA_SLOW_RET_CMD;
      A     "HALF_SECOND_PULSE_TRAIN";
      O     "DOOR_EXTRACTOR_DB".TRA_SLOW_RET_OP_CUT;
      O     "MAIN_POWER_DB".LAMP_TEST_PB;
      );
      =     "DOOR_EXTRACTOR_DB".TRA_SLOW_RET_IND;
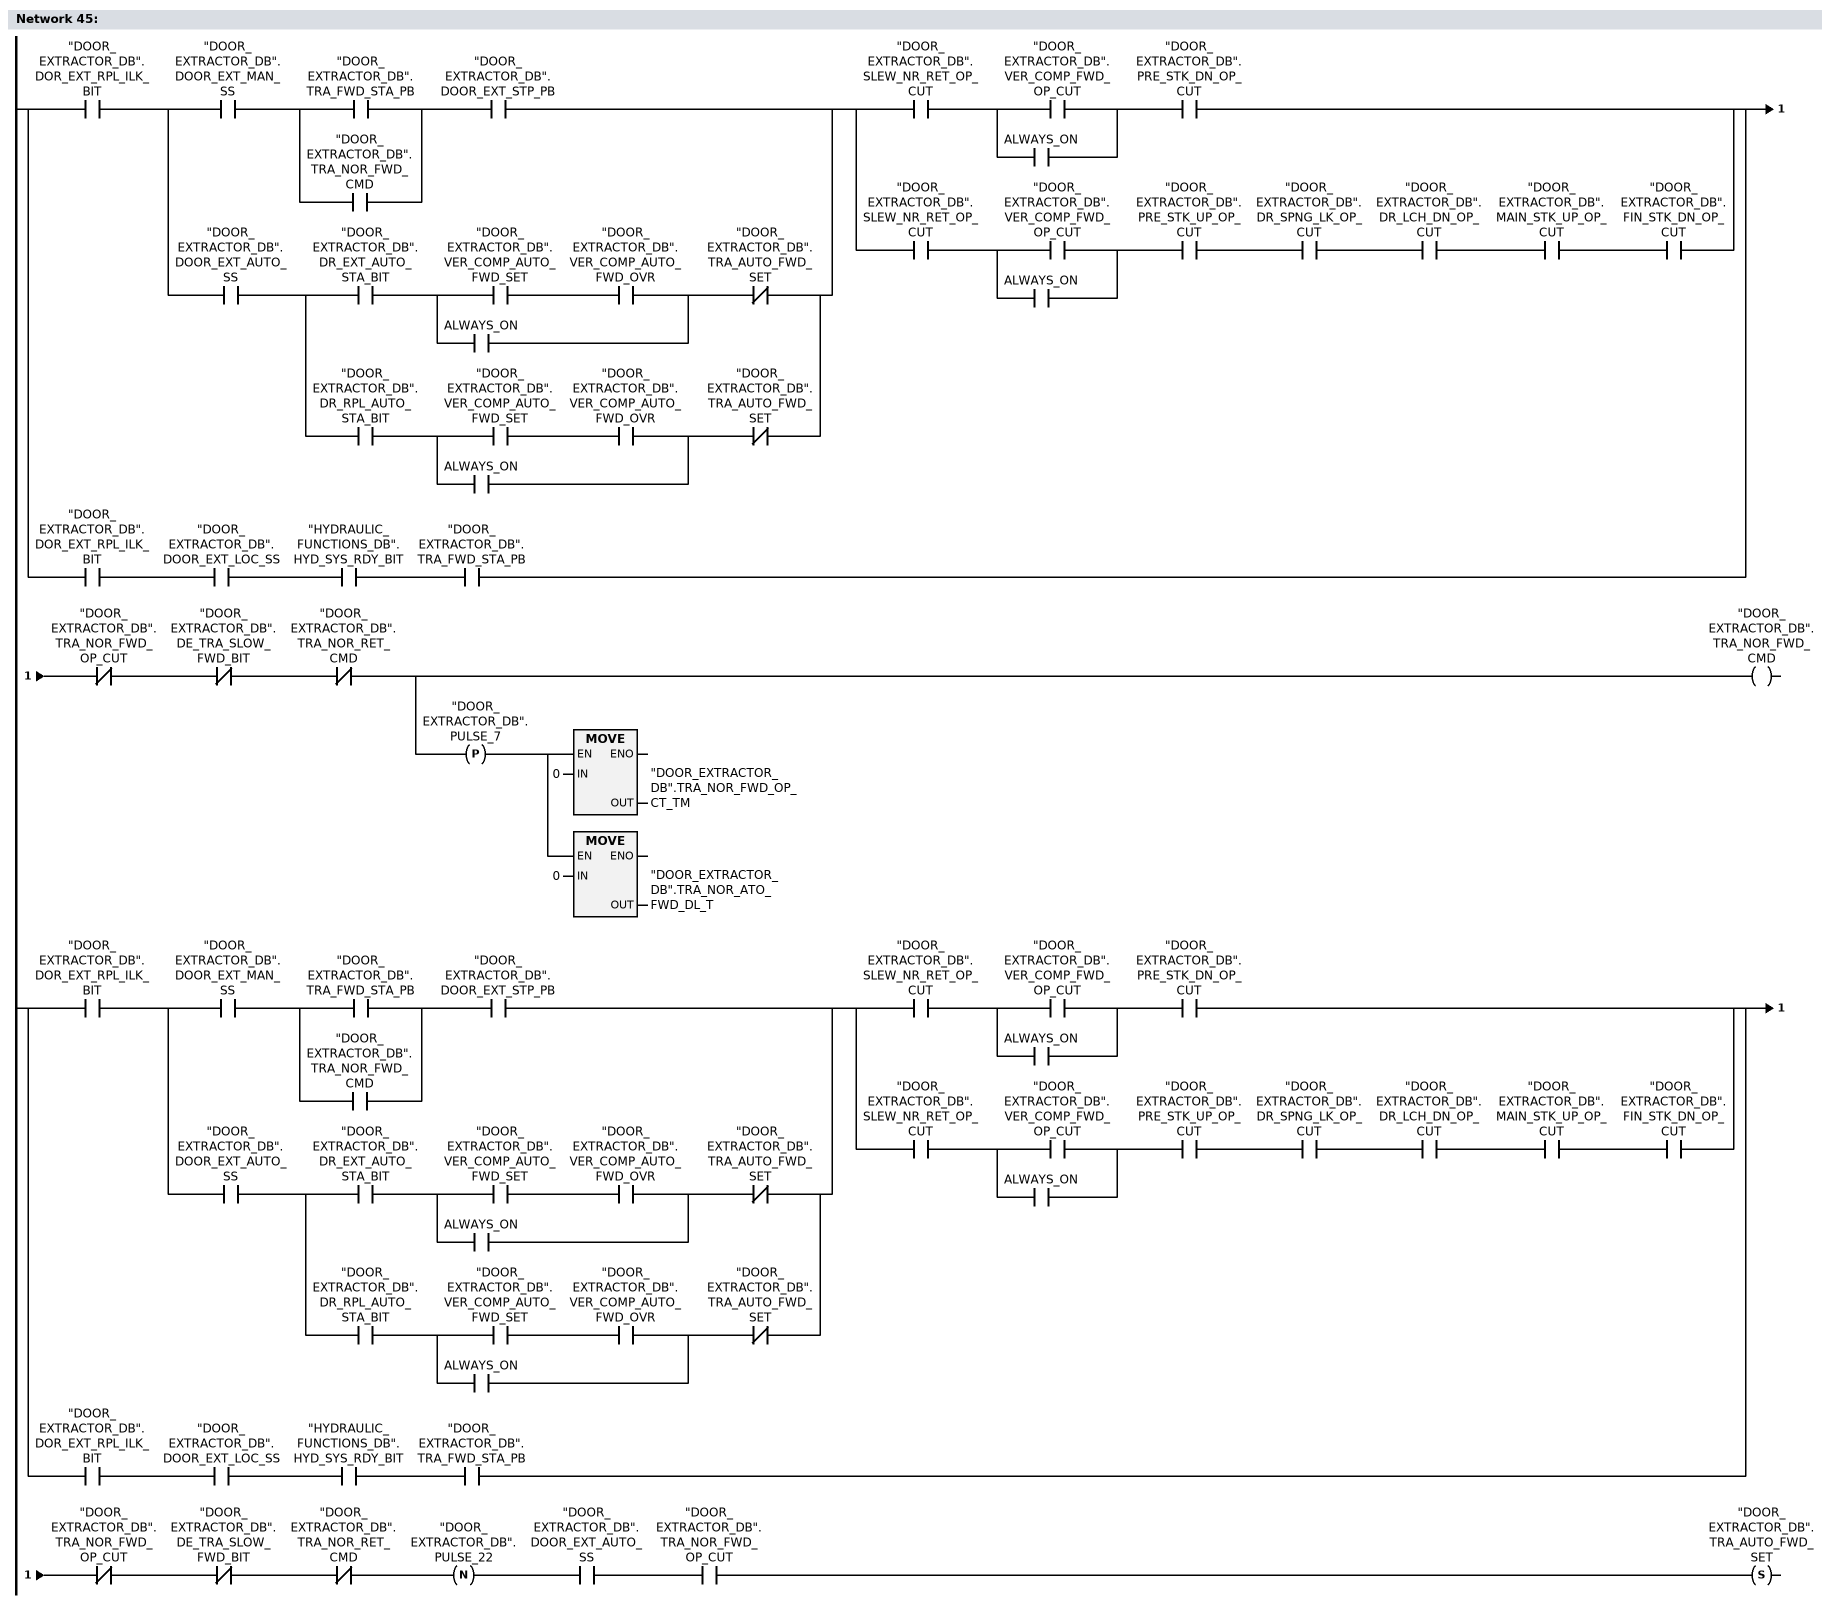
NETWORK
TITLE =
      A(;
      A     "DOOR_EXTRACTOR_DB".DOR_EXT_RPL_ILK_BIT;
      A(;
      A     "DOOR_EXTRACTOR_DB".DOOR_EXT_MAN_SS;
      A(;
      O     "DOOR_EXTRACTOR_DB".TRA_FWD_STA_PB;
      O     "DOOR_EXTRACTOR_DB".TRA_NOR_FWD_CMD;
      );
      A     "DOOR_EXTRACTOR_DB".DOOR_EXT_STP_PB;
      O;
      A     "DOOR_EXTRACTOR_DB".DOOR_EXT_AUTO_SS;
      A(;
      A     "DOOR_EXTRACTOR_DB".DR_EXT_AUTO_STA_BIT;
      A(;
      A     "DOOR_EXTRACTOR_DB".VER_COMP_AUTO_FWD_SET;
      A     "DOOR_EXTRACTOR_DB".VER_COMP_AUTO_FWD_OVR;
      O     "ALWAYS_ON";
      );
      AN    "DOOR_EXTRACTOR_DB".TRA_AUTO_FWD_SET;
      O;
      A     "DOOR_EXTRACTOR_DB".DR_RPL_AUTO_STA_BIT;
      A(;
      A     "DOOR_EXTRACTOR_DB".VER_COMP_AUTO_FWD_SET;
      A     "DOOR_EXTRACTOR_DB".VER_COMP_AUTO_FWD_OVR;
      O     "ALWAYS_ON";
      );
      AN    "DOOR_EXTRACTOR_DB".TRA_AUTO_FWD_SET;
      );
      );
      A(;
      A     "DOOR_EXTRACTOR_DB".SLEW_NR_RET_OP_CUT;
      A(;
      O     "DOOR_EXTRACTOR_DB".VER_COMP_FWD_OP_CUT;
      O     "ALWAYS_ON";
      );
      A     "DOOR_EXTRACTOR_DB".PRE_STK_DN_OP_CUT;
      O;
      A     "DOOR_EXTRACTOR_DB".SLEW_NR_RET_OP_CUT;
      A(;
      O     "DOOR_EXTRACTOR_DB".VER_COMP_FWD_OP_CUT;
      O     "ALWAYS_ON";
      );
      A     "DOOR_EXTRACTOR_DB".PRE_STK_UP_OP_CUT;
      A     "DOOR_EXTRACTOR_DB".DR_SPNG_LK_OP_CUT;
      A     "DOOR_EXTRACTOR_DB".DR_LCH_DN_OP_CUT;
      A     "DOOR_EXTRACTOR_DB".MAIN_STK_UP_OP_CUT;
      A     "DOOR_EXTRACTOR_DB".FIN_STK_DN_OP_CUT;
      );
      O;
      A     "DOOR_EXTRACTOR_DB".DOR_EXT_RPL_ILK_BIT;
      A     "DOOR_EXTRACTOR_DB".DOOR_EXT_LOC_SS;
      A     "HYDRAULIC_FUNCTIONS_DB".HYD_SYS_RDY_BIT;
      A     "DOOR_EXTRACTOR_DB".TRA_FWD_STA_PB;
      );
      AN    "DOOR_EXTRACTOR_DB".TRA_NOR_FWD_OP_CUT;
      AN    "DOOR_EXTRACTOR_DB".DE_TRA_SLOW_FWD_BIT;
      AN    "DOOR_EXTRACTOR_DB".TRA_NOR_RET_CMD;
      =     L 0.0;
      A     L 0.0;
      BLD   102;
      =     "DOOR_EXTRACTOR_DB".TRA_NOR_FWD_CMD;
      A(;
      A     L 0.0;
      FN    "DOOR_EXTRACTOR_DB".PULSE_22;
      );
      A     "DOOR_EXTRACTOR_DB".DOOR_EXT_AUTO_SS;
      A     "DOOR_EXTRACTOR_DB".TRA_NOR_FWD_OP_CUT;
      S     "DOOR_EXTRACTOR_DB".TRA_AUTO_FWD_SET;
      A     L 0.0;
      FP    "DOOR_EXTRACTOR_DB".PULSE_7;
      =     L 0.1;
      A     L 0.1;
      JNB   M039;
      L     0;
      T     "DOOR_EXTRACTOR_DB".TRA_NOR_FWD_OP_CT_TM;
M039: NOP   0;
      A     L 0.1;
      JNB   M040;
      L     0;
      T     "DOOR_EXTRACTOR_DB".TRA_NOR_ATO_FWD_DL_T;
M040: NOP   0;
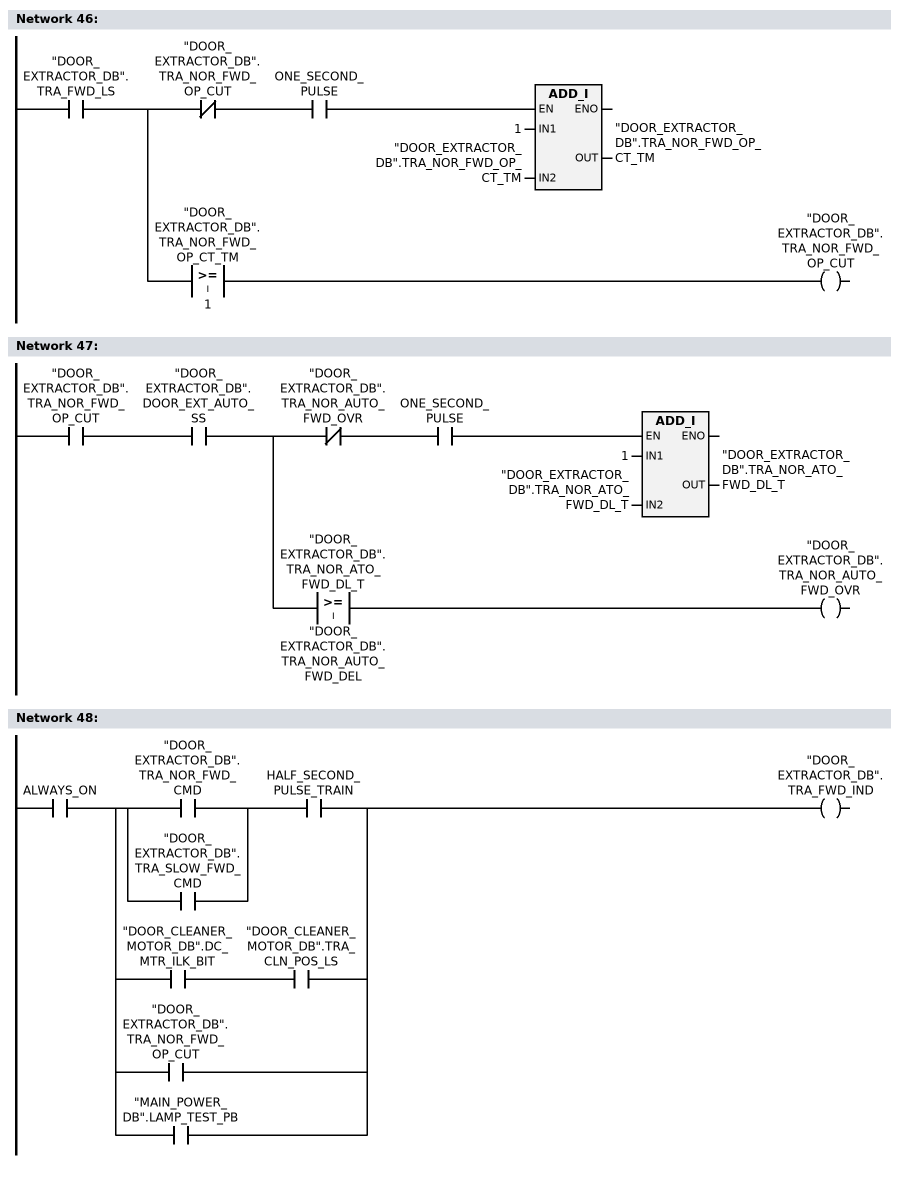
NETWORK
TITLE =
      A     "DOOR_EXTRACTOR_DB".TRA_FWD_LS;
      =     L 0.0;
      A     L 0.0;
      AN    "DOOR_EXTRACTOR_DB".TRA_NOR_FWD_OP_CUT;
      A     "ONE_SECOND_PULSE";
      JNB   M041;
      L     1;
      L     "DOOR_EXTRACTOR_DB".TRA_NOR_FWD_OP_CT_TM;
      +I;
      T     "DOOR_EXTRACTOR_DB".TRA_NOR_FWD_OP_CT_TM;
M041: NOP   0;
      A     L 0.0;
      A(;
      L     "DOOR_EXTRACTOR_DB".TRA_NOR_FWD_OP_CT_TM;
      L     1;
      >=I;
      );
      =     "DOOR_EXTRACTOR_DB".TRA_NOR_FWD_OP_CUT;
NETWORK
TITLE =
      A     "DOOR_EXTRACTOR_DB".TRA_NOR_FWD_OP_CUT;
      A     "DOOR_EXTRACTOR_DB".DOOR_EXT_AUTO_SS;
      =     L 0.0;
      A     L 0.0;
      AN    "DOOR_EXTRACTOR_DB".TRA_NOR_AUTO_FWD_OVR;
      A     "ONE_SECOND_PULSE";
      JNB   M042;
      L     1;
      L     "DOOR_EXTRACTOR_DB".TRA_NOR_ATO_FWD_DL_T;
      +I;
      T     "DOOR_EXTRACTOR_DB".TRA_NOR_ATO_FWD_DL_T;
M042: NOP   0;
      A     L 0.0;
      A(;
      L     "DOOR_EXTRACTOR_DB".TRA_NOR_ATO_FWD_DL_T;
      L     "DOOR_EXTRACTOR_DB".TRA_NOR_AUTO_FWD_DEL;
      >=I;
      );
      =     "DOOR_EXTRACTOR_DB".TRA_NOR_AUTO_FWD_OVR;
NETWORK
TITLE =
      A     "ALWAYS_ON";
      A(;
      A(;
      O     "DOOR_EXTRACTOR_DB".TRA_NOR_FWD_CMD;
      O     "DOOR_EXTRACTOR_DB".TRA_SLOW_FWD_CMD;
      );
      A     "HALF_SECOND_PULSE_TRAIN";
      O;
      A     "DOOR_CLEANER_MOTOR_DB".DC_MTR_ILK_BIT;
      A     "DOOR_CLEANER_MOTOR_DB".TRA_CLN_POS_LS;
      O     "DOOR_EXTRACTOR_DB".TRA_NOR_FWD_OP_CUT;
      O     "MAIN_POWER_DB".LAMP_TEST_PB;
      );
      =     "DOOR_EXTRACTOR_DB".TRA_FWD_IND;
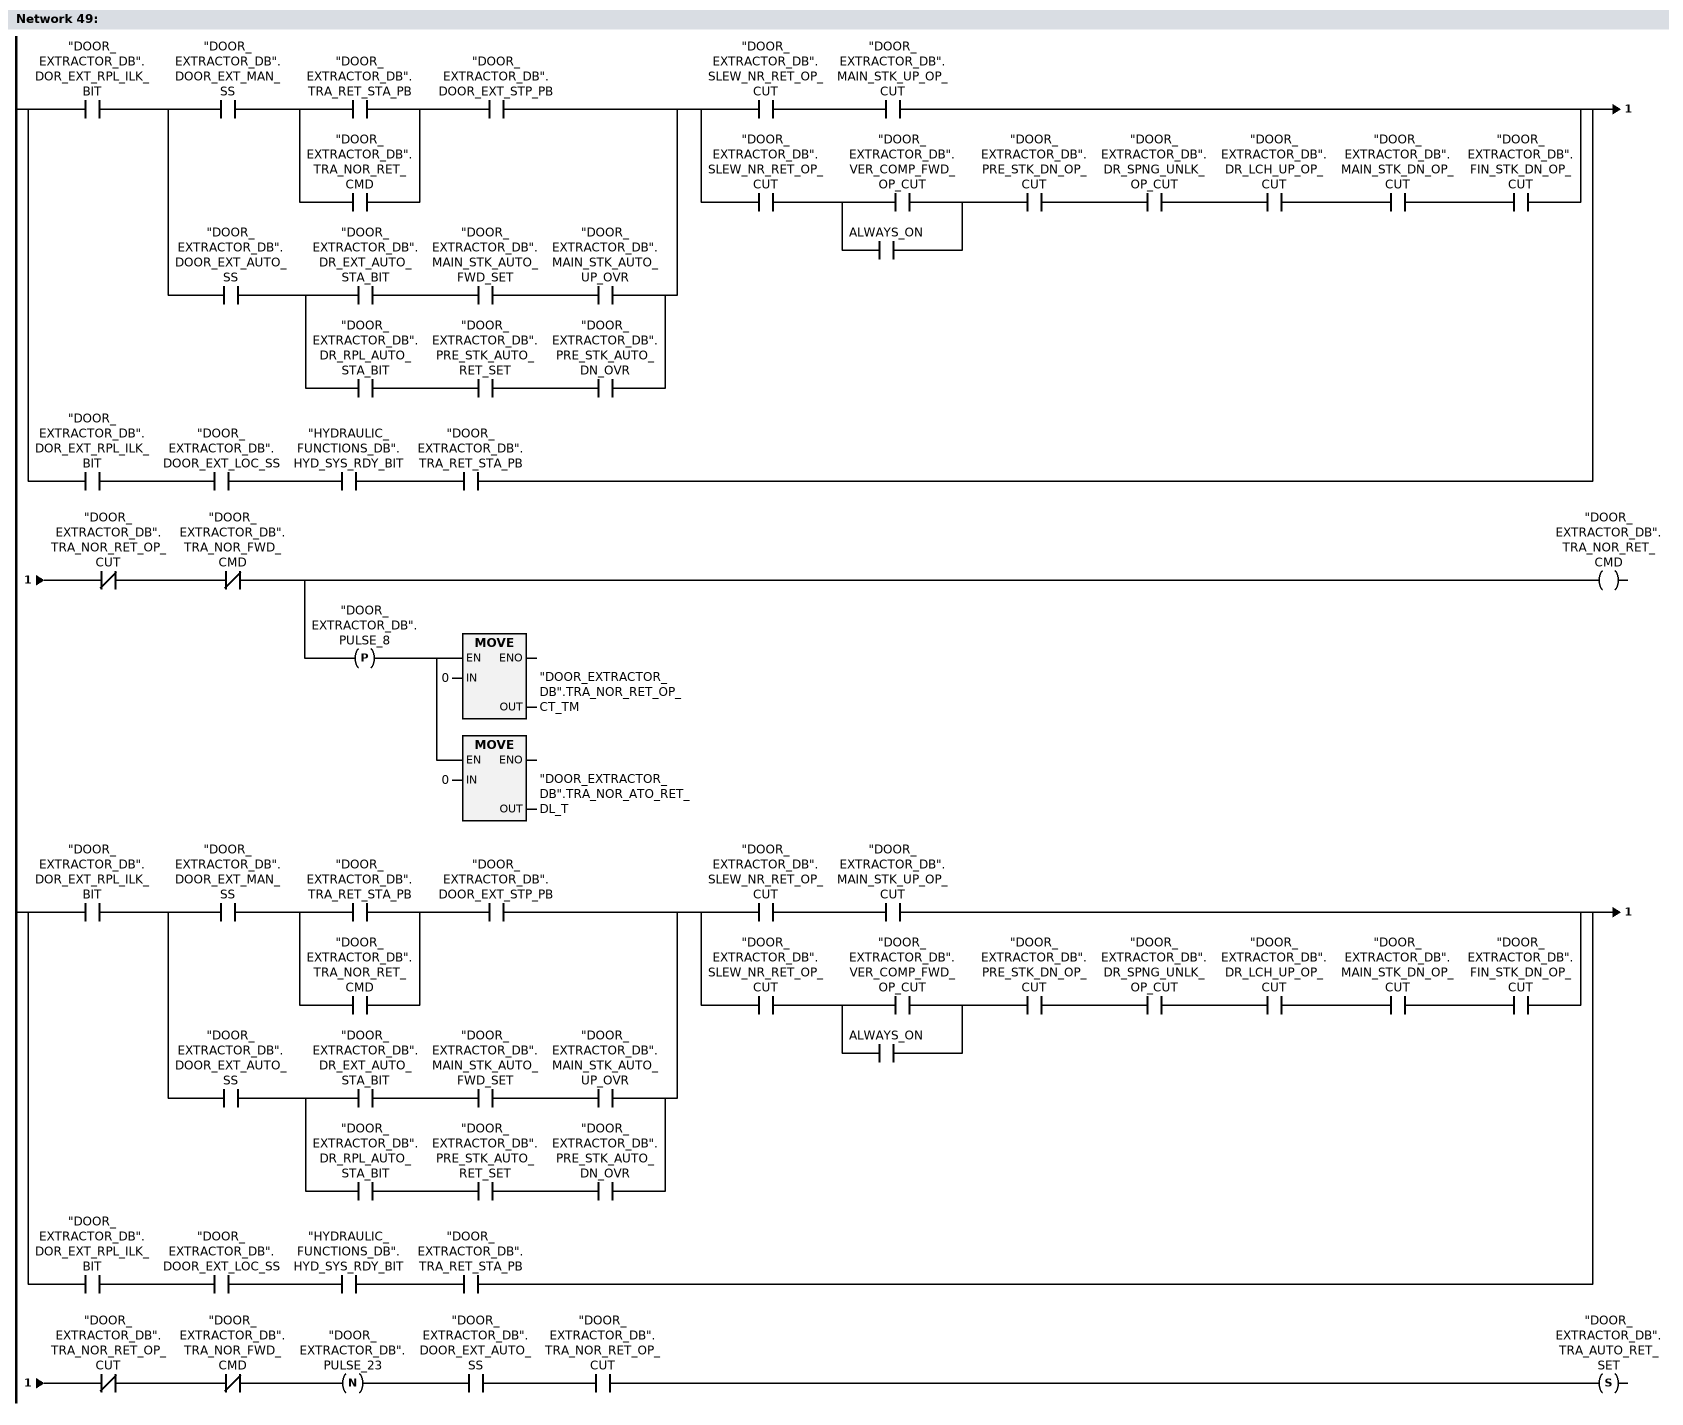
NETWORK
TITLE =
      A(;
      A     "DOOR_EXTRACTOR_DB".DOR_EXT_RPL_ILK_BIT;
      A(;
      A     "DOOR_EXTRACTOR_DB".DOOR_EXT_MAN_SS;
      A(;
      O     "DOOR_EXTRACTOR_DB".TRA_RET_STA_PB;
      O     "DOOR_EXTRACTOR_DB".TRA_NOR_RET_CMD;
      );
      A     "DOOR_EXTRACTOR_DB".DOOR_EXT_STP_PB;
      O;
      A     "DOOR_EXTRACTOR_DB".DOOR_EXT_AUTO_SS;
      A(;
      A     "DOOR_EXTRACTOR_DB".DR_EXT_AUTO_STA_BIT;
      A     "DOOR_EXTRACTOR_DB".MAIN_STK_AUTO_FWD_SET;
      A     "DOOR_EXTRACTOR_DB".MAIN_STK_AUTO_UP_OVR;
      O;
      A     "DOOR_EXTRACTOR_DB".DR_RPL_AUTO_STA_BIT;
      A     "DOOR_EXTRACTOR_DB".PRE_STK_AUTO_RET_SET;
      A     "DOOR_EXTRACTOR_DB".PRE_STK_AUTO_DN_OVR;
      );
      );
      A(;
      A     "DOOR_EXTRACTOR_DB".SLEW_NR_RET_OP_CUT;
      A     "DOOR_EXTRACTOR_DB".MAIN_STK_UP_OP_CUT;
      O;
      A     "DOOR_EXTRACTOR_DB".SLEW_NR_RET_OP_CUT;
      A(;
      O     "DOOR_EXTRACTOR_DB".VER_COMP_FWD_OP_CUT;
      O     "ALWAYS_ON";
      );
      A     "DOOR_EXTRACTOR_DB".PRE_STK_DN_OP_CUT;
      A     "DOOR_EXTRACTOR_DB".DR_SPNG_UNLK_OP_CUT;
      A     "DOOR_EXTRACTOR_DB".DR_LCH_UP_OP_CUT;
      A     "DOOR_EXTRACTOR_DB".MAIN_STK_DN_OP_CUT;
      A     "DOOR_EXTRACTOR_DB".FIN_STK_DN_OP_CUT;
      );
      O;
      A     "DOOR_EXTRACTOR_DB".DOR_EXT_RPL_ILK_BIT;
      A     "DOOR_EXTRACTOR_DB".DOOR_EXT_LOC_SS;
      A     "HYDRAULIC_FUNCTIONS_DB".HYD_SYS_RDY_BIT;
      A     "DOOR_EXTRACTOR_DB".TRA_RET_STA_PB;
      );
      AN    "DOOR_EXTRACTOR_DB".TRA_NOR_RET_OP_CUT;
      AN    "DOOR_EXTRACTOR_DB".TRA_NOR_FWD_CMD;
      =     L 0.0;
      A     L 0.0;
      BLD   102;
      =     "DOOR_EXTRACTOR_DB".TRA_NOR_RET_CMD;
      A(;
      A     L 0.0;
      FN    "DOOR_EXTRACTOR_DB".PULSE_23;
      );
      A     "DOOR_EXTRACTOR_DB".DOOR_EXT_AUTO_SS;
      A     "DOOR_EXTRACTOR_DB".TRA_NOR_RET_OP_CUT;
      S     "DOOR_EXTRACTOR_DB".TRA_AUTO_RET_SET;
      A     L 0.0;
      FP    "DOOR_EXTRACTOR_DB".PULSE_8;
      =     L 0.1;
      A     L 0.1;
      JNB   M043;
      L     0;
      T     "DOOR_EXTRACTOR_DB".TRA_NOR_RET_OP_CT_TM;
M043: NOP   0;
      A     L 0.1;
      JNB   M044;
      L     0;
      T     "DOOR_EXTRACTOR_DB".TRA_NOR_ATO_RET_DL_T;
M044: NOP   0;
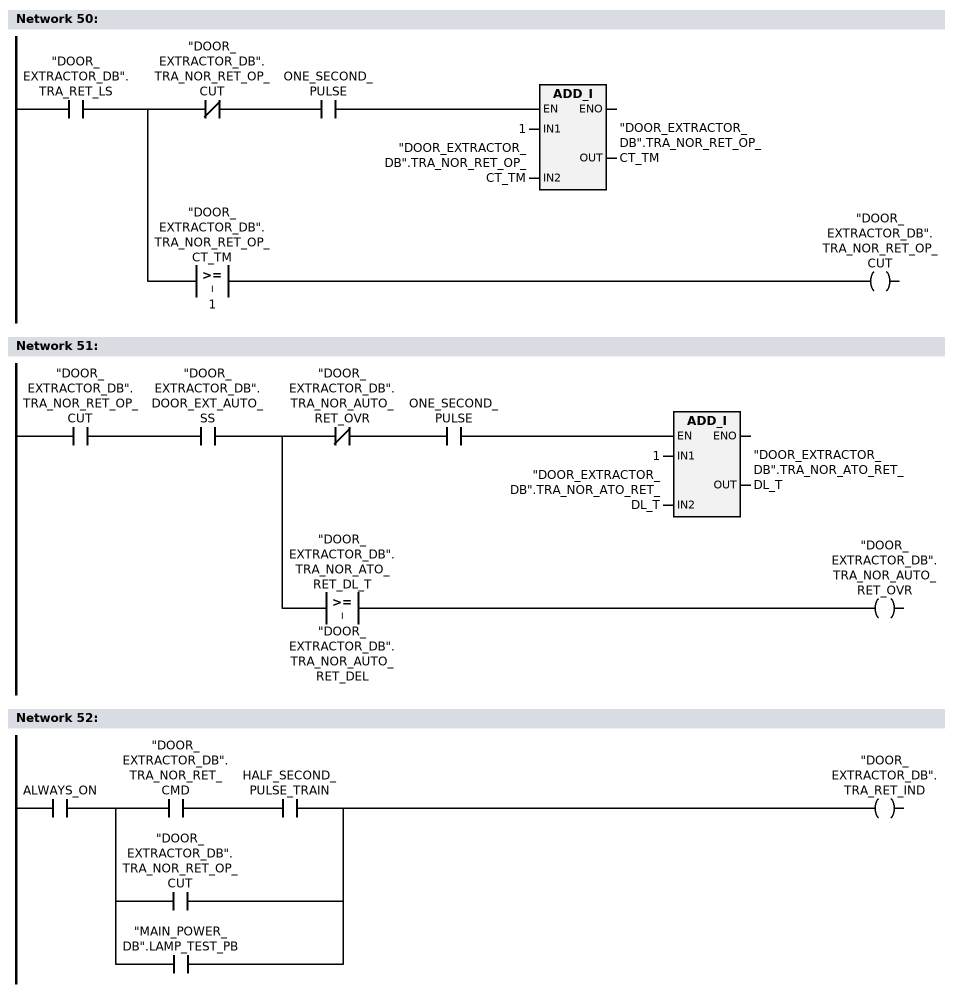
NETWORK
TITLE =
      A     "DOOR_EXTRACTOR_DB".TRA_RET_LS;
      =     L 0.0;
      A     L 0.0;
      AN    "DOOR_EXTRACTOR_DB".TRA_NOR_RET_OP_CUT;
      A     "ONE_SECOND_PULSE";
      JNB   M045;
      L     1;
      L     "DOOR_EXTRACTOR_DB".TRA_NOR_RET_OP_CT_TM;
      +I;
      T     "DOOR_EXTRACTOR_DB".TRA_NOR_RET_OP_CT_TM;
M045: NOP   0;
      A     L 0.0;
      A(;
      L     "DOOR_EXTRACTOR_DB".TRA_NOR_RET_OP_CT_TM;
      L     1;
      >=I;
      );
      =     "DOOR_EXTRACTOR_DB".TRA_NOR_RET_OP_CUT;
NETWORK
TITLE =
      A     "DOOR_EXTRACTOR_DB".TRA_NOR_RET_OP_CUT;
      A     "DOOR_EXTRACTOR_DB".DOOR_EXT_AUTO_SS;
      =     L 0.0;
      A     L 0.0;
      AN    "DOOR_EXTRACTOR_DB".TRA_NOR_AUTO_RET_OVR;
      A     "ONE_SECOND_PULSE";
      JNB   M046;
      L     1;
      L     "DOOR_EXTRACTOR_DB".TRA_NOR_ATO_RET_DL_T;
      +I;
      T     "DOOR_EXTRACTOR_DB".TRA_NOR_ATO_RET_DL_T;
M046: NOP   0;
      A     L 0.0;
      A(;
      L     "DOOR_EXTRACTOR_DB".TRA_NOR_ATO_RET_DL_T;
      L     "DOOR_EXTRACTOR_DB".TRA_NOR_AUTO_RET_DEL;
      >=I;
      );
      =     "DOOR_EXTRACTOR_DB".TRA_NOR_AUTO_RET_OVR;
NETWORK
TITLE =
      A     "ALWAYS_ON";
      A(;
      A     "DOOR_EXTRACTOR_DB".TRA_NOR_RET_CMD;
      A     "HALF_SECOND_PULSE_TRAIN";
      O     "DOOR_EXTRACTOR_DB".TRA_NOR_RET_OP_CUT;
      O     "MAIN_POWER_DB".LAMP_TEST_PB;
      );
      =     "DOOR_EXTRACTOR_DB".TRA_RET_IND;
